	20: // wait reading PAI info completed
		fbCoeReadPAIInfo.bExecute := FALSE;
		IF NOT fbCoeReadPAIInfo.bBusy THEN
			M_UpdateError(fbCoeReadPAIInfo.bError, fbCoeReadPAIInfo.nErrId);
			nStepGetPAIInfo := 0;
		END_IF
END_CASE

fbCoeReadPAIInfo(
	sNetId:= F_CreateAmsNetId(stAdsAddr.netId), 
	nSlaveAddr:= nSlaveAddress, 
	nSubIndex:= 1, 
	nIndex:= nIdxPAIInfo, 
	pDstBuf:= ADR(stPAIInfoData), 
	cbBufLen:= SIZEOF(stPAIInfoData),
	bCompleteAccess:= TRUE);
END_METHOD

METHOD PRIVATE M_WfGetSlaveState : BOOL
// workflow read slave state
CASE nStepGetState OF
	0: // idle
	
	10: // start reading actual slave state
		fbGetSlaveState.bExecute := TRUE;
		nStepGetState := 20;
		
	20: // wait reading actual slave state completed
		fbGetSlaveState.bExecute := FALSE;
		IF NOT fbGetSlaveState.bBusy THEN
			M_UpdateError(fbGetSlaveState.bError, fbGetSlaveState.nErrId);
			IF NOT fbGetSlaveState.bError THEN
				stSlaveState := F_ConvSlaveStateToBitsEx(fbGetSlaveState.state);
			END_IF			
			nStepGetState := 0;				
		END_IF
END_CASE

fbGetSlaveState(
	sNetId := F_CreateAmsNetId(stAdsAddr.netId), 
	nSlaveAddr := nSlaveAddress);
END_METHOD

END_FUNCTION_BLOCK

// ---- POUs/System/Utilities/Convert/F_EcDeviceTimeStampToTime.TcPOU
FUNCTION F_EcDeviceTimeStampToTime : TIME
VAR_INPUT
	nDeviceTimeStamp : ULINT;
END_VAR
VAR
	fDevieTimeStamp : LREAL;
END_VAR

fDevieTimeStamp := ULINT_TO_LREAL(nDeviceTimeStamp) / 1E6; 		// ns to ms
F_EcDeviceTimeStampToTime := LREAL_TO_TIME(fDevieTimeStamp);	// ms to time

END_FUNCTION

// ---- POUs/System/Recipe/FB_RecipeManager.TcPOU
FUNCTION_BLOCK FB_RecipeManager
VAR_IN_OUT	
	/// Recipe	            
	stRecipe	: ST_Settings;
	
	/// Logger
	nLogger		: I_Logger;
	
	/// PlcTag Browser
	fbVar2File	: FB_Var2File;
END_VAR
VAR_INPUT
	/// Directory of recipe files
	sRecipePath					:T_MaxString := '/usr/local/var2file/data/';
	
	/// Allows to load a recipe (Machine is stopped)
	bEnableLoadRecipe			:BOOL;
END_VAR
VAR_OUTPUT
	/// Loading/Saving busy
	bBusy						:BOOL;
	bLoadingBusy				:BOOL;
	stActiveRecipeName			:ST_Text;
	/// Error
	bError						:BOOL;
	stErrorText					:ST_Text;
END_VAR
VAR
	sFileExtension				:STRING := '.csv';
	sObjectNameRecipe			:STRING(255) := 'Services.fbRecipeManager.stRecipeWork';
	
	bInit						:BOOL;
	posSaveCurrent				:R_TRIG;
	posNewRecipe				:R_TRIG;
	posChangeRecipe				:R_TRIG;
	posRefreshRecipeList		:R_TRIG;
	posLoadRecipe				:R_TRIG;
	posDeleteRecipe				:R_TRIG;
	posCopyRecipe				:R_TRIG;

	stRecipeWork				:ST_Settings;
	
	bErrorListRecipes			:BOOL;
	bErrorLoadRecipe			:BOOL;
	bErrorSaveRecipe			:BOOL;
	bErrorCopyRecipe			:BOOL;

	stWorkText					:ST_Text;
	rtrigBusy					:R_TRIG;
END_VAR


// show current recipe data
HMI.stHmi.stOut.stCommon.stRecipe.wsActiveRecipe := stRecipe.stPlant_Settings[E_PlantSettings.ePlantSetting_RecipeName].sValue;
HMI.stHmi.stOut.stCommon.stRecipe.wsActiveRecipeComment := stRecipe.stPlant_Settings[E_PlantSettings.ePlantSetting_RecipeComment].sValue;
HMI.stHmi.stOut.stCommon.stRecipe.wsActiveRecipeProduct := stRecipe.stProduct_Settings[E_ProductSettings.eProductSettings_ProductNumber].sValue;

stActiveRecipeName := F_CreateDynText(stRecipe.stPlant_Settings[E_PlantSettings.ePlantSetting_RecipeName].sValue,0);

// Save current recipe
posSaveCurrent(CLK := stHmi.stIn.stRecipe.bSaveCurrentRecipe);
IF posSaveCurrent.Q AND NOT bBusy THEN
	// copy current
	stRecipeWork := stRecipe;
	M_SaveRecipe(TRUE);
END_IF

// Update current
posChangeRecipe(CLK := stHmi.stIn.stRecipe.bUpdateRecipe );
IF posChangeRecipe.Q THEN
	IF HMI.stHmi.stIn.stRecipe.wsNewEditRecipeName <> "" THEN
		stRecipe.stPlant_Settings[E_PlantSettings.ePlantSetting_RecipeName].sValue := stHmi.stIn.stRecipe.wsNewEditRecipeName;		
	END_IF
	stRecipe.stPlant_Settings[E_PlantSettings.ePlantSetting_RecipeComment].sValue := stHmi.stIn.stRecipe.wsNewEditRecipeComment;		
	stRecipe.stProduct_Settings[E_ProductSettings.eProductSettings_ProductNumber].sValue := stHmi.stIn.stRecipe.wsNewEditRecipeProduct;		
END_IF

// Save as new
posNewRecipe(CLK := stHmi.stIn.stRecipe.bCreateNewRecipe );
IF posNewRecipe.Q AND stHmi.stIn.stRecipe.wsNewEditRecipeName <> "" AND
NOT bBusy THEN
	// copy current
	stRecipeWork := stRecipe;
	// change
	stRecipeWork.stPlant_Settings[E_PlantSettings.ePlantSetting_RecipeName].sValue := stHmi.stIn.stRecipe.wsNewEditRecipeName;		
	stRecipeWork.stPlant_Settings[E_PlantSettings.ePlantSetting_RecipeComment].sValue := stHmi.stIn.stRecipe.wsNewEditRecipeComment;		
	stRecipeWork.stProduct_Settings[E_ProductSettings.eProductSettings_ProductNumber].sValue := stHmi.stIn.stRecipe.wsNewEditRecipeProduct;		
	M_SaveRecipe(TRUE);
END_IF

// refresh list of recipes
posRefreshRecipeList(CLK := stHmi.stIn.stRecipe.bRefreshRecipeList OR NOT bInit);
IF posRefreshRecipeList.Q THEN
	M_ListRecipes(TRUE);
END_IF


// Load
posLoadRecipe(CLK := stHmi.stIn.stRecipe.bLoadSelectedRecipe);
IF posLoadRecipe.Q AND NOT bBusy THEN
	IF stHmi.stIn.stRecipe.nSelectedRecipe >= 0 AND stHmi.stIn.stRecipe.nSelectedRecipe <= CONST.iMaxIdxRecipe AND_THEN 
	HMI.stHmi.stOut.stCommon.stRecipe.aRecipeList[stHmi.stIn.stRecipe.nSelectedRecipe] <> "" THEN
		M_LoadRecipe(TRUE, HMI.stHmi.stOut.stCommon.stRecipe.aRecipeList[stHmi.stIn.stRecipe.nSelectedRecipe]);
	END_IF
END_IF

// delete
posDeleteRecipe(CLK := stHmi.stIn.stRecipe.bDeleteSelectedRecipe);
IF posDeleteRecipe.Q THEN
	IF stHmi.stIn.stRecipe.nSelectedRecipe >= 0 AND stHmi.stIn.stRecipe.nSelectedRecipe <= CONST.iMaxIdxRecipe AND_THEN 
	HMI.stHmi.stOut.stCommon.stRecipe.aRecipeList[stHmi.stIn.stRecipe.nSelectedRecipe] <> "" THEN
		M_DeleteRecipe(TRUE, HMI.stHmi.stOut.stCommon.stRecipe.aRecipeList[stHmi.stIn.stRecipe.nSelectedRecipe]);
	END_IF	
END_IF

// copy
posCopyRecipe(CLK := stHmi.stIn.stRecipe.bCopySelectedRecipe);
IF posCopyRecipe.Q AND NOT bBusy THEN
	IF stHmi.stIn.stRecipe.nSelectedRecipe >= 0 AND stHmi.stIn.stRecipe.nSelectedRecipe <= CONST.iMaxIdxRecipe AND_THEN 
	HMI.stHmi.stOut.stCommon.stRecipe.aRecipeList[stHmi.stIn.stRecipe.nSelectedRecipe] <> "" AND
	stHmi.stIn.stRecipe.wsCopyRecipeNewName <> "" THEN
		M_CopyRecipe(TRUE, 
					HMI.stHmi.stOut.stCommon.stRecipe.aRecipeList[stHmi.stIn.stRecipe.nSelectedRecipe],
					stHmi.stIn.stRecipe.wsCopyRecipeNewName);
	END_IF		
END_IF


// calls
M_SaveRecipe(FALSE);
M_ListRecipes(FALSE);
M_LoadRecipe(FALSE, "");
M_DeleteRecipe(FALSE, "");
M_CopyRecipe(FALSE, "", "");

// Supervision
M_Supervision();

// show HMI Status fields
rtrigBusy(CLK := bBusy);
IF rtrigBusy.Q THEN
	HMI.stHmi.stOut.stCommon.stRecipe.bStatusTextVisible := TRUE; // show immediately
END_IF

IF bError THEN
	HMI.stHmi.stOut.stCommon.stRecipe.stStatusText := stErrorText;
	HMI.stHmi.stOut.stCommon.stRecipe.stStatusColor.color := F_ColorToStringHexColor(STATICS.stColor.Red);
	HMI.stHmi.stOut.stCommon.stRecipe.bStatusTextVisible := TRUE;
	
ELSIF bBusy THEN
	HMI.stHmi.stOut.stCommon.stRecipe.stStatusText := stWorkText;
	HMI.stHmi.stOut.stCommon.stRecipe.stStatusColor.color := F_ColorToStringHexColor(STATICS.stColor.Blue);
	IF Statics.stPulse.bImpulse1000ms THEN
		HMI.stHmi.stOut.stCommon.stRecipe.bStatusTextVisible := NOT HMI.stHmi.stOut.stCommon.stRecipe.bStatusTextVisible;	
	END_IF

ELSE
	HMI.stHmi.stOut.stCommon.stRecipe.bStatusTextVisible := FALSE;
	HMI.stHmi.stOut.stCommon.stRecipe.stStatusText := F_CreateDynText("",0);
	
END_IF


// Enable HMI actions
HMI.stHmi.stOut.stCommon.stRecipe.bEnableSaveCurrentRecipe := NOT bBusy AND HMI.stHmi.stOut.stCommon.stRecipe.wsActiveRecipe <> "";

HMI.stHmi.stOut.stCommon.stRecipe.bEnableCreateNewRecipe := NOT bBusy AND stHmi.stIn.stRecipe.wsNewEditRecipeName <> "";
HMI.stHmi.stOut.stCommon.stRecipe.bEnableUpdateRecipe := NOT bBusy AND stHmi.stIn.stRecipe.wsNewEditRecipeName <> "";

// valid index?
IF stHmi.stIn.stRecipe.nSelectedRecipe >= 0 AND stHmi.stIn.stRecipe.nSelectedRecipe <= CONST.iMaxIdxRecipe THEN
	HMI.stHmi.stOut.stCommon.stRecipe.bEnableLoadRecipe := bEnableLoadRecipe AND
																	NOT bBusy AND 
																	HMI.stHmi.stOut.stCommon.stRecipe.aRecipeList[stHmi.stIn.stRecipe.nSelectedRecipe] <> "";
	HMI.stHmi.stOut.stCommon.stRecipe.bEnableDeleteRecipe := NOT bBusy AND 
																	(HMI.eUserLevel >= E_User_Level.eUser_Level_Maintenance) AND
																	HMI.stHmi.stOut.stCommon.stRecipe.aRecipeList[stHmi.stIn.stRecipe.nSelectedRecipe] <> "" AND
																	HMI.stHmi.stOut.stCommon.stRecipe.aRecipeList[stHmi.stIn.stRecipe.nSelectedRecipe] <> HMI.stHmi.stOut.stCommon.stRecipe.wsActiveRecipe;
	HMI.stHmi.stOut.stCommon.stRecipe.bEnableCopyRecipe := NOT bBusy AND 
																	HMI.stHmi.stOut.stCommon.stRecipe.aRecipeList[stHmi.stIn.stRecipe.nSelectedRecipe] <> "";	
ELSE
	HMI.stHmi.stOut.stCommon.stRecipe.bEnableLoadRecipe := FALSE;
	HMI.stHmi.stOut.stCommon.stRecipe.bEnableDeleteRecipe := FALSE;
	HMI.stHmi.stOut.stCommon.stRecipe.bEnableCopyRecipe := FALSE;	
END_IF



bInit := TRUE;

METHOD PRIVATE M_CopyRecipe : BOOL
VAR_INPUT
	bCopyRecipe				:BOOL;
	wsRecipeName_From		:WSTRING(255);
	wsRecipeName_To			:WSTRING(255);
END_VAR
VAR_INST
	wsRecipeName_FromWork		:WSTRING(255);
	wsRecipeName_ToWork			:WSTRING(255);
	wsRecipeName_ToWork_noExt	:WSTRING(255); //Recipename without FileExtension
	nStep				:INT;
END_VAR

// Reset error
IF HMI.stHmi.stIn.stMain.stButton_Reset.bClick THEN
	bErrorCopyRecipe := FALSE;
END_IF

IF nStep > 0 THEN
	stWorkText := F_CreateDynText("Rezept wird kopiert...",0);
END_IF

CASE nStep OF
	
	0:
		IF bCopyRecipe AND wsRecipeName_From <> "" AND
		wsRecipeName_To <> "" AND NOT fbVar2File.bBusy THEN
			wsRecipeName_FromWork := wsRecipeName_From;
			wsRecipeName_ToWork := wsRecipeName_To;
			wsRecipeName_ToWork_noExt := wsRecipeName_ToWork;
			bErrorCopyRecipe := FALSE;
			bBusy := TRUE;
			nStep := 100;
		END_IF
		
		
		// LOAD

		// load recipe over var2file to stRecipeWork and save it with a new name
		// add sFileExtension ('.csv') to the filename
	100:
		wsRecipeName_FromWork := WCONCAT2x(wsRecipeName_FromWork, TO_WSTRING(sFileExtension));
		wsRecipeName_ToWork := WCONCAT2x(wsRecipeName_ToWork, TO_WSTRING(sFileExtension));
		// copy current for none recipe settings
		stRecipeWork := stRecipe;
		// Load to work
		fbVar2File.M_LoadFromFileRecipe(sRecipePath, TO_STRING(wsRecipeName_FromWork));
		nStep := 110;
		
	110:
		IF fbVar2File.bBusy THEN
			nStep := 120;	
		END_IF
		
	120:
		IF fbVar2File.bError THEN
			bErrorCopyRecipe := TRUE;
			nStep := 200;
			
		ELSIF fbVar2File.bDone THEN
			nStep := 150;
			
		END_IF
		
		
		// SAVE
	150:	
		stRecipeWork.stPlant_Settings[E_PlantSettings.ePlantSetting_RecipeName].sValue := wsRecipeName_ToWork_noExt;
		// Trigger save action
		fbVar2File.M_SaveToFileRecipe(sObjectNameRecipe,
			sRecipePath, TO_STRING(wsRecipeName_ToWork) );
		nStep := 160;
		
	160:
		IF fbVar2File.bBusy THEN
			nStep := 170;	
		END_IF
		
	170:
		IF fbVar2File.bError THEN
			bErrorCopyRecipe := TRUE;
			nStep := 200;
			
		ELSIF fbVar2File.bDone THEN
			nStep := 200;
			
		END_IF
			
	200:
		bBusy := FALSE;
		nStep := 0;
		M_ListRecipes(TRUE);
		
END_CASE
END_METHOD

METHOD PRIVATE M_DeleteRecipe : BOOL
VAR_INPUT
	bDeleteRecipe			:BOOL;
	wsRecipeName			:WSTRING(255);
END_VAR
VAR_INST
	wsRecipeNameWork		:WSTRING(255);
	nStep					:INT;
	fbDeleteFile			:FB_FileDelete;
	
END_VAR

fbDeleteFile.sNetId := '';

IF nStep > 0 THEN
	stWorkText := F_CreateDynText("Rezept wird gelöscht...",0);
END_IF

CASE nStep OF
	
	0:
		IF bDeleteRecipe AND wsRecipeName <> "" THEN
			wsRecipeNameWork := wsRecipeName;
			bBusy := TRUE;
			nStep := 100;
		END_IF
		
		
		// delete recipe
		// add sFileExtension ('.csv') to the filename
	100:
		fbDeleteFile.sPathName := CONCAT4(sRecipePath, sDirSeparator, TO_STRING(wsRecipeNameWork), sFileExtension);
		fbDeleteFile(bExecute := FALSE);
		fbDeleteFile(bExecute := TRUE);
		IF fbDeleteFile.bBusy THEN
			nStep := 110;
		END_IF
		
	110:
		fbDeleteFile(bExecute := FALSE);
		IF NOT fbDeleteFile.bBusy THEN
			nStep := 200;		
		END_IF
		
		// finish
	200:
		bBusy := FALSE;
		nStep := 0;
		M_ListRecipes(TRUE);

END_CASE
END_METHOD

METHOD M_ListRecipes : BOOL
VAR_INPUT
	bRefreshRecipeList			:BOOL;
END_VAR
VAR_INST
	nStepRefreshRecLst			:INT;
	fbListFiles					:FB_EnumFindFileEntry;
	nFileIdx					:INT;
END_VAR

fbListFiles.sNetId := '';
fbListFiles.sPathName := CONCAT4(sRecipePath, sDirSeparator, '*', sFileExtension);

HMI.stHmi.stOut.stCommon.stRecipe.nMaxEntryRecipeList := nFileIdx;

// Reset error
IF HMI.stHmi.stIn.stMain.stButton_Reset.bClick THEN
	bErrorListRecipes := FALSE;
END_IF

CASE nStepRefreshRecLst OF
	
		// wait start
	0:
		fbListFiles( bExecute := FALSE );
		IF bRefreshRecipeList THEN
			FOR nFileIdx := 0 TO CONST.iMaxIdxRecipe DO
				HMI.stHmi.stOut.stCommon.stRecipe.aRecipeList[nFileIdx] := "";
			END_FOR
			nFileIdx := 0;
			bErrorListRecipes := FALSE;
			fbListFiles.eCmd := E_EnumCmdType.eEnumCmd_First;	
			nStepRefreshRecLst := 100;
		END_IF
		
		// Read
	100:
		fbListFiles( bExecute := FALSE );
		fbListFiles( bExecute := TRUE );
		IF fbListFiles.bBusy THEN
			nStepRefreshRecLst := 110;		
		END_IF
		
		// get value
	110:
		fbListFiles( bExecute := FALSE );
		IF NOT fbListFiles.bBusy THEN
			IF NOT fbListFiles.bError THEN
				IF NOT fbListFiles.bEOE AND nFileIdx <= CONST.iMaxIdxRecipe THEN
					// save in array
					HMI.stHmi.stOut.stCommon.stRecipe.aRecipeList[nFileIdx] := TO_WSTRING(F_Replace(fbListFiles.stFindFile.sFileName, sFileExtension, ''));
                    fbListFiles.eCmd := eEnumCmd_Next; (* enum next entry *)
					
					nFileIdx := nFileIdx + 1;
                    nStepRefreshRecLst := 100;
					
				ELSE
					nStepRefreshRecLst := 0; // finish
				END_IF
			
			ELSE
				nStepRefreshRecLst := 0;
				bErrorListRecipes := TRUE;
			END_IF
		END_IF

END_CASE
END_METHOD

METHOD PRIVATE M_LoadRecipe : BOOL
VAR_INPUT
	bLoadRecipe			:BOOL;
	wsRecipeName		:WSTRING(255);
END_VAR
VAR_INST
	wsRecipeNameWork		:WSTRING(255);
	nStep					:INT;
END_VAR

// Reset error
IF HMI.stHmi.stIn.stMain.stButton_Reset.bClick THEN
	bErrorLoadRecipe := FALSE;
END_IF

IF nStep > 0 THEN
	stWorkText := F_CreateDynText("Rezept wird geladen...",0);
END_IF

CASE nStep OF
	
	0:
	
		bLoadingBusy := FALSE;
		IF bLoadRecipe AND wsRecipeName <> "" AND NOT fbVar2File.bBusy THEN
			wsRecipeNameWork := wsRecipeName;
			bBusy := TRUE;
			bLoadingBusy := TRUE;
			bErrorLoadRecipe := FALSE;
			nStep := 100;
		END_IF
		
		
		// load recipe over var2file to stRecipeWork
	100:
		wsRecipeName := WCONCAT2x(wsRecipeNameWork, TO_WSTRING(sFileExtension));
		// copy current for none recipe settings
		stRecipeWork := stRecipe;
		// Trigger load action
		fbVar2File.M_LoadFromFileRecipe(sRecipePath, TO_STRING(wsRecipeName));
		nStep := 110;
		
	110:
		IF fbVar2File.bBusy THEN
			nStep := 120;	
		END_IF
		
	120:
		IF fbVar2File.bError THEN
			bErrorLoadRecipe := TRUE;
			nStep := 200;
			
		ELSIF fbVar2File.bDone THEN
			stRecipe := stRecipeWork; // Takeover recipe data
			nStep := 200;
			
		END_IF
				
	200:
		bBusy := FALSE;
		nStep := 0;

END_CASE
END_METHOD

METHOD M_LoadRecipeStart : BOOL
VAR_INPUT
	wsRecipeName	: WSTRING;
END_VAR
M_LoadRecipe(TRUE, wsRecipeName);
M_LoadRecipeStart := true;
END_METHOD

METHOD PRIVATE M_SaveRecipe : BOOL
VAR_INPUT
	bSaveRecipe			:BOOL;
END_VAR
VAR_INST
	nStep				:INT;
	wsRecipeName		:WSTRING(255);
END_VAR

// Reset error
IF HMI.stHmi.stIn.stMain.stButton_Reset.bClick THEN
	bErrorSaveRecipe := FALSE;
END_IF

IF nStep > 0 THEN
	stWorkText := F_CreateDynText("Rezept wird gespeichert...",0);
END_IF

CASE nStep OF
	
	0:
		wsRecipeName := stRecipeWork.stPlant_Settings[E_PlantSettings.ePlantSetting_RecipeName].sValue;
		IF bSaveRecipe AND wsRecipeName <> "" AND NOT fbVar2File.bBusy THEN
			bBusy := TRUE;
			bErrorSaveRecipe := FALSE;
			nStep := 100;
		END_IF
		
		
		// save recipe over var2file from stRecipeWork
	100:
		wsRecipeName := WCONCAT2x(wsRecipeName, TO_WSTRING(sFileExtension));
		// Trigger save action
		fbVar2File.M_SaveToFileRecipe(sObjectNameRecipe,
			sRecipePath, TO_STRING(wsRecipeName) );
		nStep := 110;
		
	110:
		IF fbVar2File.bBusy THEN
			nStep := 120;	
		END_IF
		
	120:
		IF fbVar2File.bError THEN
			bErrorSaveRecipe := TRUE;
			nStep := 200;
			
		ELSIF fbVar2File.bDone THEN
			nStep := 200;
			
		END_IF
		
	200:
		HMI.stHmi.stOut.stCommon.stRecipe.wsActiveRecipeSavedInfo := TO_WSTRING(Statics.sTimeString);
		bBusy := FALSE;
		nStep := 0;

END_CASE
END_METHOD

METHOD PRIVATE M_Supervision : BOOL
VAR_INPUT
END_VAR
// Error / Status

bError := FALSE;
stErrorText := CONST.stTextListGlobal.stText_notext;

IF bErrorListRecipes THEN
	bError := TRUE;
	stErrorText := CONST.stTextListGlobal.stText_Recipe_ListError;
	
ELSIF bErrorLoadRecipe THEN
	bError := TRUE;
	stErrorText := fbVar2File.stErrorText;
	
ELSIF bErrorSaveRecipe THEN
	bError := TRUE;
	stErrorText := fbVar2File.stErrorText;

ELSIF bErrorCopyRecipe THEN
	bError := TRUE;
	stErrorText := CONST.stTextListGlobal.stText_Recipe_CopyError;
	
END_IF
END_METHOD

END_FUNCTION_BLOCK

// ---- POUs/System/Utilities/Var2File/FB_Var2File.TcPOU
/// Handler for interact with the Var2File tool
FUNCTION_BLOCK FB_Var2File
VAR_INPUT
	stConfig			:ST_Var2File_Config;
END_VAR	
VAR_OUTPUT
	/// Fehlerzustand
	bError				:BOOL;
	/// Fehlertext
	stErrorText			:ST_Text;
	/// Fehlertext Zusatz
	stErrorText_Add		:ST_Text;
	/// Warnung
	bWarning			:BOOL;
	/// Warnungstext
	stWarnText			:ST_Text;

	bBusy		: BOOL;
	bDone		: BOOL;
	nProgress	: UDINT;
END_VAR
VAR
	// object vars
	// start load / save
	fbStart_Exe					: NT_StartProcess;
	// find file
	fbFindFile					: FB_EnumFindFileEntry;
	
	nProcessStep				: INT;

	// Com struct for application
	stAppCom					: ST_Var2File_Com;
	
	// Save to file start flag
	bStartSave2File				: BOOL;
	// load from file flag
	bStartLoadFromFile			: BOOL;
	
	nUseFiltersetId				: INT;
	sUserDynFilterString		: STRING(255);
	sUseFileFolder				: STRING(255);
	sUseFileName				: STRING(255);
	bRecipeMode					: BOOL;
	
	// path to var2file exe
	sPathString					: STRING(100);
	sWriteToPlc					: STRING(5) := 'false';
	sCommand					: T_MAXSTRING;
	
	rtrig_Error					: R_TRIG;
	
	// check communication with var2file tool
	tonCheckCom					: TON;
END_VAR

(*
Parameter:
	-	Mode:			GUI-Mode oder Background-Mode
	-	WriteToPlc:		Funktionsmodus	
		o	wenn TRUE dann werden Variablen in SPS geschrieben
		o	wenn FALSE werden variablen von der SPS in die Datei geschrieben	
	-	AMS-NetID:		Ziel NetId aus der die Variablen gelesen/geschrieben werden sollen
	-	AMS-Port:		Ziel Portnummer
	-	Filter-Set-ID:		ID (Nummer) des Filtersets das angewendet werden soll
	-	Dyn.FilterString:	Statt Filter-Set-ID kann ein Filterstring direkt übergeben werden
	-	FileFolder:		Zielordner für Export-Import Datei
	-	FileName:		Dateiname

Beispiele:
	xxxx.exe -Mode Background -amsnetid “192.168.1.1.1.1” -port 851 -filterset 3
	xxxx.exe -Mode Background -amsnetid “192.168.1.1.1.1” -port 851 -filterstring “GVL_TEST”

	Plausibilität-checks
*)

// now in TC/BSD mode!

tonCheckCom(PT := T#1M);
tonCheckCom.IN := FALSE;

CASE nProcessStep OF
	0:
		// reset data
		IF bStartSave2File OR bStartLoadFromFile THEN
			// reset communication structure
			MEMSET(ADR(stAppCom), 0, SIZEOF(stAppCom));
			
			M_Reset();
			fbStart_Exe.START := FALSE;
			fbFindFile.bExecute := FALSE;
			
			M_CheckPlausibility();
			
			// build path string to exe
			sPathString := CONCAT( stConfig.sAppExeFilePath, stConfig.sAppExeFileName);
		END_IF
		
		// start sequence
		IF bStartSave2File THEN
			sWriteToPlc := 'false';
			bStartSave2File := FALSE;
			nProcessStep := 10; // save data
		ELSIF bStartLoadFromFile THEN
			sWriteToPlc := 'true';
			bStartLoadFromFile := FALSE;
			nProcessStep := 50; // load data
		END_IF
		
// save data
	10: 
		// build command string
		IF stConfig.sAmsNetId = '' THEN
			sCommand := CONCAT4(sPathString, 
						' -mode background ',
						'',
						' -port 851 ');						
		ELSE
			sCommand := CONCAT4(sPathString, 
						' -mode background -amsNetId "',
						stConfig.sAmsNetId,
						'" -port 851 ');			
		END_IF

		// add filter
		IF nUseFiltersetId <> 0 THEN
			sCommand := CONCAT3(sCommand, 
						' -filterSet ',
						INT_TO_STRING(nUseFiltersetId));
		ELSE
			sCommand := CONCAT4(sCommand, 
						' -filterstring "',
						sUserDynFilterString,
						'"');
		END_IF
		
		// recipe mode
		IF bRecipeMode THEN
			sCommand := CONCAT3(sCommand, 
						' -recipe true ',
						'');			
		END_IF
				
		// add file destination
		sCommand := CONCAT5(sCommand, 
					' -filePath "',
					sUseFileFolder,
					'" -fileName ',
					sUseFileName);
	
		nProcessStep := 100;
		
// load data
	50: // enum first entry
		fbFindFile.eCmd := eEnumCmd_First;
		nProcessStep := 60;
		
	60: // start search file
		fbFindFile(bExecute := FALSE);
		fbFindFile(bExecute := TRUE);
		nProcessStep := 70;
		
	70: // wait search is done
		fbFindFile.bExecute := FALSE;
		IF NOT fbFindFile.bBusy THEN
			IF NOT fbFindFile.bError THEN
				// File found
				IF fbFindFile.stFindFile.sFileName = sUseFileName THEN
					nProcessStep := 80;
					
				// End of file reached -> file not found
				ELSIF fbFindFile.bEOE THEN
					bError := TRUE;
					stErrorText := F_CreateDynText(TO_WSTRING(CONCAT(sUseFileName, ' - file not found!')), 0);
				
					bBusy := FALSE;
					nProcessStep := 0;
					
				// search next file
				ELSE
					fbFindFile.eCmd := eEnumCmd_Next; // enum next entry 
					nProcessStep := 60;
				END_IF
				
			// log error
			ELSE
				bError := TRUE;
				stErrorText := F_CreateDynText(TO_WSTRING(CONCAT(sUseFileName, ' - file or directory not found!')), 0);
							
				bBusy := FALSE;
				nProcessStep := 0;
			END_IF
		END_IF

	80: 
		// build command string
		IF stConfig.sAmsNetId = '' THEN
			sCommand := CONCAT4(sPathString, 
						' -mode background -writeToPlc true ',
						'',
						' -port 851 ');		
		ELSE
			sCommand := CONCAT4(sPathString, 
						' -mode background -writeToPlc true -amsNetId "',
						stConfig.sAmsNetId,
						'" -port 851 ');			
		END_IF
		
		// recipe mode
		IF bRecipeMode THEN
			sCommand := CONCAT3(sCommand, 
						' -recipe true ',
						'');			
		END_IF
			
		// add file destination
		sCommand := CONCAT6(sCommand, 
					' -filePath "',
					sUseFileFolder,
					'" -fileName "',
					sUseFileName,
					'"');
					
		nProcessStep := 100;

// start application and check communication with tool

	100: // execute app
		fbStart_Exe.START := TRUE;
		// wait busy
		IF fbStart_Exe.BUSY THEN
			fbStart_Exe.START := FALSE;
			nProcessStep := 110;
		END_IF
		
	110: // wait not busy
		IF NOT fbStart_Exe.BUSY THEN
			IF fbStart_Exe.ERR THEN
				bBusy := FALSE;
				nProcessStep := 0;
			ELSE
				nProcessStep := 120;
			END_IF
		END_IF
	
	120: // check communication with tool
		// tool is done
		IF stAppCom.bAppJobFinished OR stAppCom.nAppProgress = 100 THEN
			M_ErrorCode(stAppCom.nAppErrorCode);
			bBusy := FALSE;
			nProcessStep := 0;
			bRecipeMode := FALSE;
		ELSE
			tonCheckCom.IN := stAppCom.nAppProgress = 0;
		END_IF
		
		// error -> no communication
		IF tonCheckCom.Q OR stAppCom.nAppErrorCode > 0 THEN
			// create alarm
			bError := TRUE;
			stErrorText := F_CreateDynText(WCONCAT2x("Error Var2File tool. Error: ", M_ErrorCode(stAppCom.nAppErrorCode)), 0);
			bBusy := FALSE;
			nProcessStep := 0;
			bRecipeMode := FALSE;
		END_IF
		
END_CASE

// call FB's
IF nProcessStep > 0 THEN
	fbStart_Exe(
			NETID	:= '', // local
			PATHSTR	:= '/bin/sh', // now in TC/BSD mode!, sPathString,
			DIRNAME	:= '/usr/local/var2file', // stConfig.sAppExeFilePath,
			COMNDLINE := CONCAT4('ExecuteVar2File.sh ', sWriteToPlc, ' ', sUseFileName), //sCommand,
			TMOUT	:= T#5S,
			BUSY	=> , 
			ERR		=> , 
			ERRID	=> );
			
	fbFindFile(
			sNetID := '', 
			sPathName := CONCAT3(sUseFileFolder, sDirSeparator, '*.*'),
			tTimeout := T#5S);
END_IF	
						
// set alarm
rtrig_Error( CLK := fbStart_Exe.ERR);
IF rtrig_Error.Q THEN
	bError := TRUE;
	stErrorText := F_CreateDynText(WCONCAT2x("Var2File NT_Process ErrorID: ", TO_WSTRING(fbStart_Exe.ERRID)), 0);
END_IF

bDone := stAppCom.bAppJobFinished AND NOT bBusy;
nProgress := stAppCom.nAppProgress;

			
(*// call FB's (nur Backup hier)
fbStart_Var2File(
			NETID	:= '', 
			PATHSTR	:= 'C:\Rmth\Software\var2file\var2file.exe',//'C:\Tools\var2file_Rmth\PlcTag.WinForms.App.exe', //sPathString, 
			DIRNAME	:= 'C:\Rmth\Software\var2file',//'C:\Tools\var2file_Rmth', //WSTRING_TO_STRING(wsUseFileFolder), 
			COMNDLINE := 'C:\Rmth\Software\var2file\var2file.exe -mode background -amsNetId "192.168.163.1.1.1" -port 851 -filterSet 1 -filePath "C:\Temp" -fileName PlcData.json', 
			TMOUT	:= T#5S,
			BUSY	=> , 
			ERR		=> , 
			ERRID	=> );*)

METHOD PROTECTED M_CheckPlausibility : BOOL
VAR_INPUT
END_VAR
VAR
	bPlausible			: BOOL;
	nLastBackslashPos	: INT;
END_VAR
// set marker bit
bPlausible := FALSE;

// plausibility check
IF stConfig.sAppExeFilePath = '' THEN
	bError := TRUE;
	stErrorText := F_CreateDynText("No Var2File exe path", 0);
	
ELSIF stConfig.sAppExeFileName = '' THEN
	bError := TRUE;
	stErrorText := F_CreateDynText("No Var2File exe name", 0);
	
ELSIF sUseFileFolder = '' THEN
	bError := TRUE;
	stErrorText := F_CreateDynText("No file folder selected (Var2File)", 0);
	
ELSIF sUseFileName = '' THEN
	bError := TRUE;
	stErrorText := F_CreateDynText("No file name selected (Var2File)", 0);
	
ELSE
	bPlausible := TRUE;
	
	// check if there is 'no' backslash at the end of the file directory path
	IF RIGHT(sUseFileFolder, 1) = sDirSeparator THEN
		nLastBackslashPos := LEN(sUseFileFolder);
		sUseFileFolder := DELETE(sUseFileFolder, 1, nLastBackslashPos);
	END_IF
	
	// no point found in the filename (assumption no file extension)
	IF FIND(sUseFileName, '.') = 0 THEN
		// add file extension .json
		sUseFileName := CONCAT(sUseFileName, '.json');
	END_IF
	
	// check if there is a backslash at the end of the exe directory path
	IF RIGHT(stConfig.sAppExeFilePath, 1) <> sDirSeparator THEN
		stConfig.sAppExeFilePath := CONCAT(stConfig.sAppExeFilePath, sDirSeparator);
	END_IF
END_IF

IF NOT bPlausible THEN
	// reset start signals
	bStartSave2File := FALSE;
	bStartLoadFromFile := FALSE;
	bBusy := FALSE;
END_IF

M_CheckPlausibility := TRUE;
END_METHOD

/// convert Var2File error code into an text and send alarm
METHOD PRIVATE M_ErrorCode : WSTRING
VAR_INPUT
	/// Applications error code
	nErrorCode			: UDINT;
END_VAR

CASE nErrorCode OF
	0:	// No error
		RETURN;
		
	100:
		M_ErrorCode := "Job canceled by plc";
		
	101:
		M_ErrorCode := "Job canceled by operator";
		
	1000:
		M_ErrorCode := "Reading plc tags failed";
		
	1001:
		M_ErrorCode := "Reading plc tag values failed";
		
	1002:
		M_ErrorCode := "Reading backup file failed";
		
	1003:
		M_ErrorCode := "Writing backup file failed";
		
	1004:
		M_ErrorCode := "Writing plc tag values failed";
		
	ELSE
		M_ErrorCode := WCONCAT2x("Undefined error code: Error ID = ", TO_WSTRING(nErrorCode));
END_CASE

// create alarm
bError := TRUE;
END_METHOD

/// cancel active job
METHOD M_JobCancel : BOOL
VAR_INPUT
END_VAR

// not allowed if not running
IF nProcessStep <= 0 THEN
	RETURN;
END_IF

stAppCom.bJobCancelRequest := TRUE;
END_METHOD

/// Starts the var2file tool with the given file name
METHOD M_LoadFromFile : BOOL
VAR_INPUT
	sFileName					: STRING(255);	
END_VAR
// not allowed if already running
IF bBusy THEN
	M_LoadFromFile := FALSE;
	RETURN;
END_IF

M_LoadFromFile := M_LoadFromFileEx(stConfig.sDefaultFileFolderPath, sFileName);
END_METHOD

/// Starts the var2file tool with the given file folder and name
METHOD M_LoadFromFileEx : BOOL
VAR_INPUT
	sFileFolder					: STRING(255);
	sFileName					: STRING(255);	
END_VAR
// not allowed if already running
IF bBusy THEN
	M_LoadFromFileEx := FALSE;
	RETURN;
END_IF

nUseFiltersetId := 0;
sUserDynFilterString := '';

sUseFileFolder	:= sFileFolder;
sUseFileName := sFileName;

bStartLoadFromFile := TRUE;

bBusy := TRUE;

M_LoadFromFileEx := TRUE;
END_METHOD

/// Starts the var2file tool with the given file folder and name
METHOD M_LoadFromFileRecipe : BOOL
VAR_INPUT
	sFileFolder					: STRING(255);
	sFileName					: STRING(255);	
END_VAR
// not allowed if already running
IF bBusy THEN
	M_LoadFromFileRecipe := FALSE;
	RETURN;
END_IF

nUseFiltersetId := 0;
sUserDynFilterString := '';

sUseFileFolder	:= sFileFolder;
sUseFileName := sFileName;
bRecipeMode := TRUE;

bStartLoadFromFile := TRUE;

bBusy := TRUE;

M_LoadFromFileRecipe := TRUE;
END_METHOD

METHOD M_Reset : BOOL
VAR_INPUT
END_VAR
/// Fehlerzustand
bError := FALSE;
/// Fehlertext
stErrorText := CONST.stTextListGlobal.stText_notext;
/// Fehlertext Zusatz
stErrorText_Add	:= CONST.stTextListGlobal.stText_notext;
/// Warnung
bWarning := FALSE;
/// Warnungstext
stWarnText := CONST.stTextListGlobal.stText_notext;
END_METHOD

/// Starts the var2file tool for all user variables
METHOD M_SaveToFileAll : BOOL
VAR_INPUT
	sFileName					: STRING(255);	
END_VAR
// not allowed if already running
IF bBusy THEN
	M_SaveToFileAll := FALSE;
	RETURN;
END_IF

M_SaveToFileAll := M_SaveToFileFilterSetEx(stConfig.nFilterSetIDAllVars, stConfig.sDefaultFileFolderPath, sFileName);
END_METHOD

/// Starts the var2file tool with the given filterset
METHOD M_SaveToFileFilterSet : BOOL
VAR_INPUT
	nFiltersetId				: INT;
	sFileName					: STRING(255);	
END_VAR
// not allowed if already running
IF bBusy THEN
	M_SaveToFileFilterSet := FALSE;
	RETURN;
END_IF

M_SaveToFileFilterSet := M_SaveToFileFilterSetEx(nFiltersetId, stConfig.sDefaultFileFolderPath, sFileName);
END_METHOD

/// Starts the var2file tool with the given filterset
METHOD M_SaveToFileFilterSetEx : BOOL
VAR_INPUT
	nFiltersetId				: INT;
	sFileFolder					: STRING(255);
	SFileName					: STRING(255);	
END_VAR
// not allowed if already running
IF bBusy OR nFiltersetId = 0 THEN
	M_SaveToFileFilterSetEx := FALSE;
	RETURN;
END_IF

nUseFiltersetId := nFiltersetId;
sUserDynFilterString := '';
bRecipeMode := FALSE;

sUseFileFolder	:= sFileFolder;
sUseFileName := sFileName;

bStartSave2File := TRUE;

bBusy := TRUE;

M_SaveToFileFilterSetEx := TRUE;
END_METHOD

/// Starts the var2file tool with the given filterstring
METHOD M_SaveToFileFilterString : BOOL
VAR_INPUT
	sDynFilterString			: STRING(255);
	sFileName					: STRING(255);	
END_VAR
// not allowed if already running
IF bBusy THEN
	M_SaveToFileFilterString := FALSE;
	RETURN;
END_IF

M_SaveToFileFilterString := M_SaveToFileFilterStringEx(sDynFilterString, stConfig.sDefaultFileFolderPath, sFileName);
END_METHOD

/// Starts the var2file tool with the given filterstring
METHOD M_SaveToFileFilterStringEx : BOOL
VAR_INPUT
	sDynFilterString			: STRING(255);
	sFileFolder					: STRING(255);
	sFileName					: STRING(255);	
END_VAR
// not allowed if already running
IF bBusy OR sDynFilterString = '' THEN
	M_SaveToFileFilterStringEx := FALSE;
	RETURN;
END_IF

nUseFiltersetId := 0;
sUserDynFilterString := sDynFilterString;
bRecipeMode := FALSE;

sUseFileFolder	:= sFileFolder;
sUseFileName := sFileName;

bStartSave2File := TRUE;

bBusy := TRUE;

M_SaveToFileFilterStringEx := TRUE;
END_METHOD

METHOD M_SaveToFileRecipe : BOOL
VAR_INPUT
	sDynFilterString			: STRING(255) := 'Objects.fbRecipeManager.stRecipe.stRecipeWork';
	sFileFolder					: STRING(255);
	sFileName					: STRING(255);	
END_VAR
// not allowed if already running
IF bBusy OR sDynFilterString = '' THEN
	M_SaveToFileRecipe := FALSE;
	RETURN;
END_IF

nUseFiltersetId := 0;
sUserDynFilterString := sDynFilterString;
bRecipeMode := TRUE;

sUseFileFolder	:= sFileFolder;
sUseFileName := sFileName;

bStartSave2File := TRUE;

bBusy := TRUE;

M_SaveToFileRecipe := TRUE;
END_METHOD

END_FUNCTION_BLOCK

// ---- POUs/System/Utilities/String/WConcat2x.TcPOU
FUNCTION WConcat2x : WSTRING(255)
VAR_INPUT
	wsExpression1: WSTRING(255);
	wsExpression2: WSTRING(255);
END_VAR

WConcat2x := WCONCAT(wsExpression1, wsExpression2);

END_FUNCTION

// ---- POUs/System/Utilities/String/F_Replace.TcPOU
FUNCTION F_Replace : STRING(255)
VAR_INPUT
	sInputText		:STRING(255);
	sSearchText		:STRING(255);
	sReplaceText	:STRING(255);
END_VAR
VAR
	idxFnd			:INT;
	iLength			:INT;
END_VAR

idxFnd := FIND(sInputText, sSearchText);
iLength := LEN(sSearchText);

IF idxFnd > 0 THEN
	F_Replace := REPLACE(sInputText, sReplaceText, iLength, idxFnd);
ELSE
	F_Replace := sInputText;
END_IF

END_FUNCTION

// ---- POUs/Plant/M001_Module/FB_M001_Module.TcPOU
FUNCTION_BLOCK FB_M001_Module EXTENDS FB_ModuleBase
VAR
	// module components

	
	// actor UIs, access to: iStatus, fPosition, iVisibleState, ..
	
	// IO ref
	stIO			: REFERENCE TO ST_M001_IO;
	
	// instannce var's
	
	

END_VAR

/// 
/// Module 001 function block 
///

METHOD PRIVATE GetHgCmd_Default : ST_St030_Command
VAR
	result : ST_St030_Command;
END_VAR
// get next job for handling
// 1. drop existing HG pallet
// 2/3. put empty pallet to storage 1/2
// 4/5. put unfinished pallet to storage 1/2

// chk HG has active command
IF Plant.stSt030IHandling.ActiveCommand.Command <> E_St030_Command.eSt030_Command_none THEN
	// sb.Set('wait for active HG command done. Active cmd: ')
		//	 .Append(TO_String(Plant.stSt030IHandling.ActiveCommand.Command));
	RETURN;
END_IF
	
// prio 1: put handling command (e.g. drop existing pallet)
result := GetHgCmd_Default_Put();
IF result.Command <> E_St030_Command.eSt030_Command_none THEN
	// sb.Set('wait for requested HG command is active, cmd: ')
		//	 .Append(TO_String(Plant.stSt030IHandling.CommandRequest.Command));
	GetHgCmd_Default := result;
	RETURN;
END_IF

// prio 2-6: get handling command (e.g. get unfinished pallet)
result := GetHgCmd_Default_Get();
GetHgCmd_Default := result;
END_METHOD

METHOD PRIVATE GetHgCmd_Default_Get : ST_St030_Command
VAR
	none	: ST_St030_Command;
END_VAR
// default logic
GetHgCmd_Default_Get := none;

// chk pallet already on handling
IF Plant.stSt030IHandling.Pallet.CarrierPresent THEN
	RETURN;
END_IF

// prio 2: req empty carrier @ storage #1
IF Plant.stSt050IMould.bReqS1Empty AND 
NOT Plant.stSt040IStorage.Pallet1.HasEmptyWorkpieceplaces THEN
	IF Plant.stSt040IStorage.Pallet1.CarrierPresent THEN
		GetHgCmd_Default_Get := GetHgCmd_StorageGet(1); // 1st, get pallet from storage 1
	ELSE
		// sb.Set('wait for oven 1/2 has empty pallet)
		GetHgCmd_Default_Get := GetHgCmd_OvenGetEmptyPallet(); // get empty pallet from oven A/B
	END_IF
	RETURN;
END_IF

// prio 3: req empty carrier @ storage #2
IF Plant.stSt050IMould.bReqS2Empty AND 
NOT Plant.stSt040IStorage.Pallet2.HasEmptyWorkpieceplaces THEN
	IF Plant.stSt040IStorage.Pallet2.CarrierPresent THEN
		GetHgCmd_Default_Get := GetHgCmd_StorageGet(2); // 1st, get pallet from storage 2
	ELSE
		// sb.Set('wait for oven 1/2 has empty pallet)
		GetHgCmd_Default_Get := GetHgCmd_OvenGetEmptyPallet(); // get empty pallet from oven A/B
	END_IF
	RETURN;
END_IF

// prio 4: req unfinished carrier @ storage #1
IF Plant.stSt050IMould.bReqS1Unfinished AND 
NOT Plant.stSt040IStorage.Pallet1.HasWorkpiecesWithRequestStatus THEN
	IF Plant.stSt040IStorage.Pallet1.CarrierPresent THEN
		GetHgCmd_Default_Get := GetHgCmd_StorageGet(1); // 1st, get pallet from storage 1
	ELSE
		// sb.Set('wait for oven 1/2 has unfinished pallet)
		GetHgCmd_Default_Get := GetHgCmd_OvenGetUnfinishedPallet(); // get unfinished pallet from oven A/B
	END_IF
	RETURN;
END_IF

// prio 5: req unfinished carrier @ storage #2
IF Plant.stSt050IMould.bReqS2Unfinished AND 
NOT Plant.stSt040IStorage.Pallet2.HasWorkpiecesWithRequestStatus THEN
	IF Plant.stSt040IStorage.Pallet2.CarrierPresent THEN
		GetHgCmd_Default_Get := GetHgCmd_StorageGet(2); // 1st, get pallet from storage 2
	ELSE
		// sb.Set('wait for oven 1/2 has unfinished pallet)
		GetHgCmd_Default_Get := GetHgCmd_OvenGetUnfinishedPallet(); // get unfinished pallet from oven A/B
	END_IF
	RETURN;
END_IF

// prio 6: req no carrier @ storage #1/2
IF (Plant.stSt050IMould.bReqS1NoCarrier OR Plant.stM001IModule.bEmptyPlant) AND Plant.stSt040IStorage.Pallet1.CarrierPresent THEN
	GetHgCmd_Default_Get := GetHgCmd_StorageGet(1); // empty plant, get pallet from storage 1
ELSIF (Plant.stSt050IMould.bReqS2NoCarrier OR Plant.stM001IModule.bEmptyPlant) AND Plant.stSt040IStorage.Pallet2.CarrierPresent THEN
	GetHgCmd_Default_Get := GetHgCmd_StorageGet(2); // empty plant, get pallet from storage 2
END_IF
END_METHOD

METHOD PRIVATE GetHgCmd_Default_Put : ST_St030_Command
VAR
	none,
	result	: ST_St030_Command;
END_VAR
// default logic
GetHgCmd_Default_Put := none;

// chk pallet on handling
IF NOT Plant.stSt030IHandling.Pallet.CarrierPresent THEN
	RETURN;
END_IF

// unfinished @ hg --> to storage 1/2
IF Plant.stSt030IHandling.Pallet.HasUnfinishedWorkpieces THEN
	// sb.Set('wait for storage request unfinished')
	IF Plant.stSt050IMould.bReqS1Unfinished AND
	   NOT Plant.stSt040IStorage.Pallet1.CarrierPresent THEN
		GetHgCmd_Default_Put := GetHgCmd_StationPut(E_Station.eStation_ST040_Storage, 1);
	ELSIF Plant.stSt050IMould.bReqS2Unfinished AND
	   NOT Plant.stSt040IStorage.Pallet2.CarrierPresent THEN
		GetHgCmd_Default_Put := GetHgCmd_StationPut(E_Station.eStation_ST040_Storage, 2);
	ELSE
		// unfinished back to oven 1/2
		GetHgCmd_Default_Put := GetHgCmd_StationPut(Plant.stSt030IHandling.Source);
	END_IF
	RETURN;
END_IF

// empty @ hg --> to storage 1/2
IF Plant.stSt030IHandling.Pallet.HasEmptyWorkpieceplaces THEN
	// sb.Set('wait for storage request empty')
	IF Plant.stSt050IMould.bReqS1Empty AND
	   NOT Plant.stSt040IStorage.Pallet1.CarrierPresent THEN
		GetHgCmd_Default_Put := GetHgCmd_StationPut(E_Station.eStation_ST040_Storage, 1);
	ELSIF Plant.stSt050IMould.bReqS2Empty AND
	   NOT Plant.stSt040IStorage.Pallet2.CarrierPresent THEN
		GetHgCmd_Default_Put := GetHgCmd_StationPut(E_Station.eStation_ST040_Storage, 2);
	ELSE
		// empty back to oven 1/2
		GetHgCmd_Default_Put := GetHgCmd_StationPut(Plant.stSt030IHandling.Source);
	END_IF
	RETURN;
END_IF 

// finished & pallet full @ hg --> to oven 2
IF Plant.stSt030IHandling.Pallet.HasAllWorkpiecesFinished THEN
	// sb.Set('wait for oven 2 rdy for finished pallet)
	// full back to oven 1/2
	GetHgCmd_Default_Put := GetHgCmd_StationPut(Plant.stSt030IHandling.Source);
END_IF

//sb.Set('state not implemented: no empty/finished or unfinished');
END_METHOD

METHOD PRIVATE GetHgCmd_OvenGetEmptyPallet : ST_St030_Command
VAR
	result : ST_St030_Command;
END_VAR
result.Command := E_St030_Command.eSt030_Command_none;
IF Plant.stSt010IOvenA.Trolley.HasCarrierWithEmptyWorkpieceplace THEN
	result.Command := E_St030_Command.eSt030_Command_OvenA_Get; // get empty pallet from oven A
	result.Position := Plant.stSt010IOvenA.Trolley.SlotOfCarrierWithEmptyWorkpieceplace; 
ELSIF Plant.stSt020IOvenB.Trolley.HasCarrierWithEmptyWorkpieceplace THEN
	result.Command := E_St030_Command.eSt030_Command_OvenB_Get; // get empty pallet from oven B
	result.Position := Plant.stSt020IOvenB.Trolley.SlotOfCarrierWithEmptyWorkpieceplace;
END_IF

GetHgCmd_OvenGetEmptyPallet := result;
END_METHOD

METHOD PRIVATE GetHgCmd_OvenGetUnfinishedPallet : ST_St030_Command
VAR
	result : ST_St030_Command;
END_VAR
result.Command := E_St030_Command.eSt030_Command_none;
IF Plant.stSt010IOvenA.Trolley.HasCarrierWithUnfinishedWorkpiece THEN
	result.Command := E_St030_Command.eSt030_Command_OvenA_Get; // get unfinished pallet from oven A
	result.Position := Plant.stSt010IOvenA.Trolley.SlotOfCarrierWithUnfinishedWorkpiece;	
ELSIF Plant.stSt020IOvenB.Trolley.HasCarrierWithUnfinishedWorkpiece THEN
	result.Command := E_St030_Command.eSt030_Command_OvenB_Get; // get unfinished pallet from oven B
	result.Position := Plant.stSt020IOvenB.Trolley.SlotOfCarrierWithUnfinishedWorkpiece;
END_IF

GetHgCmd_OvenGetUnfinishedPallet := result;
END_METHOD

METHOD PRIVATE GetHgCmd_StationPut : ST_St030_Command
VAR_INPUT
	eStation 	: E_Station;
	iIxd 		: INT := 0;
END_VAR
VAR
	result 		: ST_St030_Command;
END_VAR
CASE eStation OF
	E_Station.eStation_ST010_OvenA:
		IF Plant.stSt010IOvenA.Trolley.HasEmptySlot THEN
			result.Command := E_St030_Command.eSt030_Command_OvenA_Put;
			result.Position := Plant.stSt010IOvenA.Trolley.EmptySlot;
		ELSE
			ModuleWarning.ArgSbAppend('Station has no empty slot')
				 .ArgSbAppendS(TO_STRING(eStation))
				 .ArgSetSbRaise();		
		END_IF
		
	E_Station.eStation_ST020_OvenB:
		IF Plant.stSt020IOvenB.Trolley.HasEmptySlot THEN
			result.Command := E_St030_Command.eSt030_Command_OvenB_Put;
			result.Position := Plant.stSt020IOvenB.Trolley.EmptySlot;
		ELSE
			ModuleWarning.ArgSbAppend('Station has no empty slot')
				 .ArgSbAppendS(TO_STRING(eStation))
				 .ArgSetSbRaise();	
		END_IF
		
	E_Station.eStation_ST040_Storage:
		result.Command := E_St030_Command.eSt030_Command_Storage_Put;
		result.Position := iIxd;
		
ELSE
	ModuleWarning.ArgSbAppend('Put to station not implemented! Station: ')
				 .ArgSbAppendS(TO_STRING(eStation))
				 .ArgSetSbRaise();
END_CASE

GetHgCmd_StationPut := result;
END_METHOD

METHOD PRIVATE GetHgCmd_StorageGet : ST_St030_Command
VAR_INPUT
	iIxd : INT;
END_VAR
VAR
	result : ST_St030_Command;
END_VAR
result.Command := E_St030_Command.eSt030_Command_Storage_Get;
result.Position := iIxd;

GetHgCmd_StorageGet := result;
END_METHOD

METHOD PRIVATE GetHgCmd_Type3 : ST_St030_Command
VAR
	none : ST_St030_Command;
END_VAR

// hg logic 3

GetHgCmd_Type3 := none;


// e.g.: impelemt custom handling command for type 3...
END_METHOD

METHOD PRIVATE GetHgCmd_Type5 : ST_St030_Command
VAR
	none : ST_St030_Command;
END_VAR

// hg logic 5

GetHgCmd_Type5 := none;


// e.g.: impelemt custom handling command for type 5...
END_METHOD

METHOD PRIVATE GetHgCmd_Type6 : ST_St030_Command
VAR
	none : ST_St030_Command;
END_VAR

// hg logic 6

GetHgCmd_Type6 := none;


// e.g.: impelemt custom handling command for type 6...
END_METHOD

METHOD PROTECTED M_CallObjects : BOOL
VAR
END_VAR

CALL_BVS();

// call..
END_METHOD

METHOD INTERNAL M_DynManual : BOOL
VAR_INPUT
END_VAR
IF NOT bInitManual THEN
	bInitManual := TRUE;
	MEMSET(ADR(stHmiManualOut.stObjects), 0, SIZEOF(stHmiManualOut.stObjects)); // reset
	
	//M_InitDynManualUi(fbAxisVmUi);
	
	//fbAxisVmUi.M_TargetListClear();
	//fbAxisVmUi.M_TargetListAddItem(F_CreateDynText("Home pos", 0), 15);
	//fbAxisVmUi.M_TargetListAddItem(F_CreateDynText("Pos Service", 0), 100);
END_IF
END_METHOD

METHOD PROTECTED M_DynMonitoring : BOOL
VAR_INPUT
END_VAR
M_DynMonitoring := SUPER^.M_DynMonitoring();

// init
IF NOT bInitMonitoring THEN
	bInitMonitoring := TRUE;
	MEMSET(ADR(stLocalMonitoring), 0, SIZEOF(stLocalMonitoring)); // reset
	
	M_InitDynMonitoringItem(0, 								// monitoring index 
							"VM Position", 					// name
							Name, 							// group (station name)
							E_DataType.eDataType_lreal, 	// data type							
							stTextListGlobal.stText_m);		// unit	

	M_InitDynMonitoringItem(1, "VM Geschwindigkeit", Name, E_DataType.eDataType_lreal, stTextListGlobal.stText_mmin);
END_IF

//stLocalMonitoring.astMonitoring[0].fValue := stM001IModule.fVmPos;
//stLocalMonitoring.astMonitoring[1].fValue := stM001IModule.fVmSpeed;
END_METHOD

METHOD INTERNAL M_DynSettings : BOOL
VAR_INST
	fSpeedMir : LREAL;
END_VAR
// init station settings
IF NOT bInitSettings THEN
	bInitSettings := TRUE;
	stLocalSettingsBackup := stLocalSettings; // backup
	MEMSET(ADR(stLocalSettings), 0, SIZEOF(stLocalSettings)); // reset
	
	M_InitDynSettingsItem(E_M001_Settings.eM001_Settings_Deaktiv,		// settings index
		TO_WSTRING(E_M001_Settings.eM001_Settings_Deaktiv),				// settings wsIndex
		Name,															// group
		stTextListGlobal.stText_DeactivateModule,						// name
		stTextListGlobal.stText_bool, E_DataType.eDataType_bool,		// unit & data type
		0, 1, 6);														// min, max & user level

	M_InitDynSettingsItem(E_M001_Settings.eM001_Settings_Autohome,
		TO_WSTRING(E_M001_Settings.eM001_Settings_Autohome),
		Name,
		stTextListGlobal.stText_AutoHome,
		stTextListGlobal.stText_bool, E_DataType.eDataType_bool,
		0, 1, 3);
		
//	M_InitDynSettingsItem(E_M001_Settings.eM001_Settings_PalletLayout,
//		TO_WSTRING(E_M001_Settings.eM001_Settings_PalletLayout),
//		Name,
//		F_CreateDynTextDefault("Palettenlayout (1-4)"),
//		stTextListGlobal.stText_notext, E_DataType.eDataType_int,
//		1, 4, 3);
		
	// restore values
	F_RestoreSettingValues(stLocalSettings.stDynStationSettings, stLocalSettingsBackup.stDynStationSettings);
END_IF

// run settings mgmt
//F_Settings_Management(stLocalSettings.stDynStationSettings);

// map current settings values
bAutoHome := stLocalSettings.stDynStationSettings[E_M001_Settings.eM001_Settings_Autohome].bValue;
END_METHOD

METHOD INTERNAL M_Fast : BOOL
VAR_INPUT
END_VAR
// fast task

Plant.fbSt030Handling.M_SequenceSearch();
//Plant.fbSt050Mould.M_Run();
END_METHOD

METHOD PROTECTED M_Homing
VAR
	bTmp : BOOL;
	stTmpTxt : ST_Text;
END_VAR
// Homing sequence
CASE sqHome.Step OF
	
	0:	
		sqHome.Info.Set("Warte auf GRST Start");
		IF RunStep AND NOT sqHome.InHome AND bRunHoming THEN
			bBusy := TRUE;
			sqAuto.Step := 0;
			sqHome.StartSequence()
				  .Step := 10;
		END_IF

	10:
		sqHome.Info.Set("Grundstellungsfahrt aktiv");
		IF P_Safety.bMachineRequestStop THEN
			sqHome.Info.Set("Anforderung Stop aktiv");
		ELSIF NOT P_Safety.SafetyOk THEN
			sqHome.Info.Set("Sicherheit nicht ok");
		ELSIF bRunHoming THEN
			sqHome.Step := 20;
		END_IF	
	
	20:
		sqHome.Info.Set("Warte auf Stationen in GRST");
		bTmp := TRUE;
		//FOR ii := 0 TO E_Station.eStation_nMaxIdx DO
		//	IF aIStaton[ii] = 0 THEN
		//		CONTINUE;
		//	END_IF
		//	IF NOT aIStaton[ii].InHome THEN
		//		stTmpTxt := aIStaton[ii].Name;
		//		sqHome.Info.Set("Warte auf Station in GRST: ")
		//				   .Append(stTmpTxt.wsName);
		//		bTmp := FALSE;
		//		EXIT;
		//	END_IF
		//END_FOR
		IF bTmp THEN			
			sqHome.Step := 100;
		END_IF
		
	100:
		sqHome.Info.Set("Grundstellungsfahrt aktiv");
		sqHome.Step := 1000;

	//	homing done			
	1000:
		sqHome.Info.Set("Grundstellung erreicht");
		IF sqHome.StepTime > T#1S THEN			
			bBusy := FALSE;
			sqHome.InHome := TRUE;
			bStopped := TRUE;
			bRunHoming := FALSE;
			sqAuto.Step := 0;
			sqHome.StopSequence()
				  .Step := 0;
		END_IF
END_CASE
END_METHOD

METHOD PUBLIC M_Init : IModule
VAR_INPUT
END_VAR
VAR
	IMod : IModule;
END_VAR
// set up station
ModuleNb := 1;
Module := E_Module.eModule_M001;
Name := stTextListGlobal.stText_M001_Name;

IMod := SUPER^.M_Init()
			  .M_InitEvents(TC_Events.ModuleM010EventClass.InfoEvent,
	  				  		TC_Events.ModuleM010EventClass.WarningEvent,
	  				  		TC_Events.ModuleM010EventClass.ErrorEvent);

// set up default IO references
M_SetReferences(IO.stM001_Module_IO);

// init components


P_Plant.M_RegisterModule(IMod);

bInitSettings	:= FALSE;
bInitMonitoring := FALSE;
bInitManual  	:= FALSE;

//aSClearText[EN] := 'Module init done.';
M_Init := IMod;
END_METHOD

METHOD PROTECTED M_Manual
VAR_INST
	iReq : INT;
END_VAR
// manual mode
IF (OpMode <> E_OpMode.eOpMode_manual) THEN
	RETURN;
END_IF
END_METHOD

METHOD PROTECTED M_OpModeChanged : BOOL
VAR_INPUT
END_VAR
(*bBusy := FALSE;

IF eOpMode <> E_OpMode.eOpMode_auto THEN
	sqAuto.Set(0);
END_IF*)
END_METHOD

METHOD INTERNAL M_RegisterStation : E_Module
VAR_INPUT
	Ist : IStation;
END_VAR
aIStaton[ISt.Station] := ISt;
P_Plant.M_RegisterStation(ISt);
M_RegisterStation := eModule;
END_METHOD

METHOD PUBLIC M_Run : BOOL
VAR_INPUT
END_VAR
VAR
	b1stShot				: BOOL := TRUE;
	stModuleStationsInfoRef	: REFERENCE TO ST_MODULE_STATIONS_INFO;
END_VAR
bSafetyOk := P_Safety.SafetyOk;
aIStaton[E_Station.eStation_ST010_OvenA].SafetyOk := P_Safety.SafetyOk;
aIStaton[E_Station.eStation_ST020_OvenB].SafetyOk := P_Safety.SafetyOk;
aIStaton[E_Station.eStation_ST030_Handling].SafetyOk := P_Safety.SafetyOk;
aIStaton[E_Station.eStation_ST040_Storage].SafetyOk := P_Safety.SafetyOk;
aIStaton[E_Station.eStation_ST050_Mould].SafetyOk := P_Safety.SafetyOk;

// call module base (calls station run)
M_Run := SUPER^.M_Run();

M_DynSettings();
M_DynManual();
M_DynMonitoring();

// loop module stations, collect infos
b1stShot := TRUE;
stModuleStationsInfoRef REF= stGlobalModuleInfo.astModuleStationsInfo[eModule];
FOR ii := 0 TO E_Station.eStation_nMaxIdx DO
	IF aIStaton[ii] = 0 THEN
		CONTINUE;
	END_IF
	
	F_AND_REF_EX(stModuleStationsInfoRef.bStation_All_Auto, aIStaton[ii].OpMode = E_OpMode.eOpMode_auto, b1stShot);
	F_OR_REF_EX(stModuleStationsInfoRef.bStation_Any_Step, aIStaton[ii].OpMode = E_OpMode.eOpMode_step, b1stShot);
	F_OR_REF_EX(stModuleStationsInfoRef.bStation_Any_Manual, aIStaton[ii].OpMode = E_OpMode.eOpMode_manual, b1stShot);
	
	F_OR_REF_EX(stModuleStationsInfoRef.bStation_Any_Error, aIStaton[ii].State = E_ComponentState.eComponentState_error, b1stShot);
	F_OR_REF_EX(stModuleStationsInfoRef.bStation_Any_Warning, aIStaton[ii].State = E_ComponentState.eComponentState_warning, b1stShot);
	F_OR_REF_EX(stModuleStationsInfoRef.bStation_Any_Info, aIStaton[ii].State = E_ComponentState.eComponentState_info, b1stShot);
	
	F_AND_REF_EX(stModuleStationsInfoRef.bStation_All_Started, (aIStaton[ii].OpMode = E_OpMode.eOpMode_auto OR aIStaton[ii].OpMode = E_OpMode.eOpMode_step) AND aIStaton[ii].RunCycle, b1stShot);
	F_AND_REF_EX(stModuleStationsInfoRef.bStation_All_Stopped, aIStaton[ii].Stopped, b1stShot);
	F_AND_REF_EX(stModuleStationsInfoRef.bStation_All_InHome, aIStaton[ii].InHome, b1stShot);
	F_OR_REF_EX(stModuleStationsInfoRef.bStation_Any_Homing, aIStaton[ii].Homing, b1stShot);
	
	b1stShot := FALSE;
END_FOR
END_METHOD

METHOD PROTECTED M_Sequence
VAR
END_VAR
// signal mapping (e.g.: enable)
stM001IModule.bRunCycle := RunCycle;

// automatic sequence
CASE sqAuto.Step OF
	
	0:	sqAuto.Info.Set("Warte auf Auto Start");
		IF NOT (RunCycle AND RunStep) THEN RETURN; END_IF
		
		sqAuto.Info.Set("Warte auf GRST");
		//IF sqHome.InHome AND bInHome THEN
			//fbAxisVm.SetPos(0);
			sqHome.InHome := FALSE;
			sqAuto.Step := 10;
		//ELSE
		//	INotiHdl.M_SetNotiDefaultInf(stTextlistGlobal.stText_NG_Stations, Name, stTextlistGlobal.stText_station_not_in_hp, stEmptyText);
		//END_IF
		
	10:	sqAuto.Info.Set("Prüfe Startbedingungen");
		IF NOT RunCycle THEN sqAuto.Step := 900; END_IF				
		CycleStart();		
		sqAuto.Step := 100;
		
	// work
	100: sqAuto.Info.Set("Automatik");
		TransitionLogic();
		IF NOT RunCycle THEN
			sqAuto.Step := 900;
		END_IF
		
	// stop from safety	or error
	800: sqAuto.Info.Set("Fehler/Safety Stop!");
		FOR ii := 0 TO E_Station.eStation_nMaxIdx DO
			IF aIStaton[ii] <> 0 THEN
				aIStaton[ii].RunCycle := FALSE;
			END_IF
		END_FOR
		sqAuto.Step := 900;		
		
	// rdy	
	900: sqAuto.Info.Set("Zyklus beendet");
		CycleEnd();
		sqAuto.Step := 0;

	// error
	1000: sqAuto.Info.Set("Error");
		bStopped := TRUE;
		sqHome.InHome := FALSE;
		bRunHoming := FALSE;

END_CASE
END_METHOD

METHOD INTERNAL M_SetReferences : BOOL
VAR_IN_OUT
	stIoRef : ST_M001_IO;
END_VAR
stIO REF= stIoRef;
M_SetReferences := TRUE;
END_METHOD

METHOD PROTECTED M_Supervision : BOOL
VAR_INPUT
END_VAR
// to be subclassed// chk stopped
IF NOT bRunCycle OR P_Safety.bMachineRequestStop THEN
	IF sqAuto.StepTime > T#20S THEN
		bStopped := TRUE;
	END_IF
END_IF

(*ToDo: // axis
IF fbAxisVm.bError THEN
	SUPER^.M_SetNotification(F_CreateDynTextUn(E_UniqNoti.eUniqNoti_M001_Module_ServoVm),	// id
					Name,																	// group (e.g.: station name)
					fbAxisVm.Name,															// txt1 (e.g.: source)
					fbAxisVmUi.stErrorText,													// txt2 (e.g.: error text)
					fbAxisVmUi.stBmk,														// txt3 (e.g.: BMK)
					E_AlarmPriority.Error,													// prio
					E_NotificationMode.eNotificationMode_Reset,								// notification mode
					E_AlarmStopMode.Stop);													// alarm stop mode
					

					
ELSIF NOT stIO.stIn.bCentrSuctPwrCircBreakerOk THEN
	SUPER^.M_SetNotification(F_CreateDynTextUn(E_UniqNoti.eUniqNoti_M001_CentralSuction),
					Name,
					F_CreateDynTextDefault("Fehler Netz Schutzschalter"),
					fbCentrSuction.Name,
					F_CreateDynTextDefault("BMK=+xyz-"),
					E_AlarmPriority.Error,
					E_NotificationMode.eNotificationMode_Reset,
					E_AlarmStopMode.Stop);
END_IF *)
END_METHOD

/// Reset station logic
{attribute 'object_name' := 'Reset'}
METHOD Reset
VAR
END_VAR
// base logic run
SUPER^.Reset();
END_METHOD

METHOD PRIVATE TransitionLogic : INT
VAR
	hgCmd : ST_St030_Command;
END_VAR
IF NOT Plant.stSt050IMould.bEnableHG THEN
	sqAuto.Info.Set("Wait for HG enable from mould");
	RETURN;
END_IF

// switxh logic by type
CASE Services.stSettings.stProduct_Settings[E_ProductSettings.eProductSettings_ProductType].nValue OF // or use production settings...
	3: hgCmd := GetHgCmd_Type3(); // e.g.: impelemt custom handling command for type 3...
	5: hgCmd := GetHgCmd_Type5(); // e.g.: impelemt custom handling command for type 5...
	6: hgCmd := GetHgCmd_Type6(); // e.g.: impelemt custom handling command for type 6...
ELSE
	
	// default logic
	hgCmd := GetHgCmd_Default();
END_CASE

Plant.stSt030IHandling.CommandRequest := hgCmd;
END_METHOD

END_FUNCTION_BLOCK

// ---- POUs/Plant/_Base/FB_ModuleBase.TcPOU
FUNCTION_BLOCK FB_ModuleBase EXTENDS FB_ComponentBase IMPLEMENTS IModule
VAR_INPUT
	bEmergencyStopOk 	: BOOL;
	bSafetyOk 			: BOOL;
	bEnable 			: BOOL;
	bAutoHome 			: BOOL;		// if its true station will be homed by start button
	iNumberOfStepChains	: INT := 1;	// count of stepchains per station
	iStepChainIndex		: INT; 		// index to link text of choosed stepchain to hmi
END_VAR
VAR_OUTPUT
	nStateColor			: DWORD;	// color for state of module

	bBusy				: BOOL;		// module is busy
	bTransferEnable		: BOOL;		// transfer enable from module
	stTextAuto			: ST_Text;
	stTextHome			: ST_Text;
	
	/// error-stop status
	bAutoStop_Error		: BOOL;
END_VAR
VAR
	stHmiToModule		: REFERENCE TO ST_DefaultHmiToPlc;				// default hmi to module
	stHmiManualIn		: REFERENCE TO ST_HMI_BASE_MODULE_MANUAL_IN;	// hmi manual to module
	stHmiManualOut		: REFERENCE TO ST_HMI_BASE_MODULE_MANUAL_OUT;	// hmi manual from module
	stLocalSettings		: REFERENCE TO ST_ModuleDynSettings;			// dyn. module settings
	stLocalMonitoring	: REFERENCE TO ST_Monitoring_Module;			// dyn. module monitoring
	
	stLocalSettingsBackup	: ST_ModuleDynSettings;	// dyn. module settings
	
	/// - stations of this module -
	aIStaton	: ARRAY[0..E_Station.eStation_nMaxIdx] OF IStation;
	
	nModuleNb	: INT;
	eModule		: E_Module;
	eOpMode		: E_OpMode;
	bStopped	: BOOL := TRUE;
	
	/// enable var's
	bRunCycle, bRunStep, bRunHoming, bInHome : BOOL;

	/// counter
	diCycles				: UDINT; // Zykluszähler
	diLastCycleTime			: UDINT; // letzte Zykluszeit [ms]
	
	tonOpModeOff			: TON;
	fTrigSafetyOk			: F_TRIG;
	rtrigOpModeChanged		: R_TRIG;
	
	rtirgSafetyOpMode_Auto	: R_TRIG;
	rtirgSafetyOpMode_Hand	: R_TRIG;
	rtirgSafetyOpMode_Aus	: R_TRIG;
	
	bInitSettings	: BOOL;
	bInitMonitoring	: BOOL;
	bInitManual		: BOOL;
	
	sb				: FB_StringBuilder;
	sqHome, sqAuto	: FB_SequenceHelperSb;
	localEvents		: ST_DefaultEventClasses;
END_VAR
VAR PERSISTENT
	diTotalCycles	: UDINT; // Zykluszähler
	eOpModeOld		: E_OpMode;
END_VAR

METHOD PROTECTED CycleEnd
VAR_INPUT
END_VAR
diCycles := diCycles + 1;
diTotalCycles := diTotalCycles + 1;
diLastCycleTime := TIME_TO_UDINT(sqAuto.SeqTime);
sqAuto.StopSequence();
bBusy := FALSE;
//bStopped := TRUE;
END_METHOD

METHOD PROTECTED CycleStart
VAR_INPUT
END_VAR
sqAuto.StartSequence();
bBusy := TRUE;
bStopped := FALSE;
END_METHOD

{attribute 'monitoring':='call'}
PROPERTY PUBLIC EmergencyStopOk : BOOL
GET
EmergencyStopOk := bEmergencyStopOk;
END_GET
SET
bEmergencyStopOk := EmergencyStopOk;
END_SET
END_PROPERTY

{attribute 'monitoring':='call'}
PROPERTY PUBLIC Enable : BOOL
GET
Enable := bEnable;
END_GET
SET
bEnable := Enable;
END_SET
END_PROPERTY

{attribute 'monitoring':='call'}
//{attribute 'monitoring' := 'variable'}
PROPERTY PUBLIC EnableManual : BOOL
GET
EnableManual := EnableSummary AND (eOpMode = eOpMode_manual);
END_GET
END_PROPERTY

{attribute 'monitoring':='call'}
//{attribute 'monitoring' := 'variable'}
PROPERTY INTERNAL EnableSummary : BOOL
GET // PUBLIC
EnableSummary := bEnable 
				AND bSafetyOk 
				AND (eOpMode = eOpMode_manual) OR (eOpMode = eOpMode_step) OR (eOpMode = eOpMode_auto);
END_GET
END_PROPERTY

METHOD PUBLIC GetStepChainTest : ST_Text
VAR_INPUT
	Index : INT; // step chain index
END_VAR
// step chain index is ignored in the default implementation -> if multiple step chains are needed, use derived base and override this method. 
GetStepChainTest.nNameId := sqAuto.InfoTextId;
GetStepChainTest.wsName := sqAuto.Info.ToWString();
GetStepChainTest.wsNameId := sqAuto.InfoTextWsId;
END_METHOD

/// Station in Home flag
{attribute 'monitoring':='call'}
PROPERTY InHome : BOOL
GET
InHome := TRUE;
//FOR ii := 0 TO iNumberOfStepChains - 1 DO
	IF NOT sqHome.InHome THEN
		InHome := FALSE;
	END_IF
//END_FOR

bInHome := InHome;
IF InHome THEN
	bRunHoming := FALSE;
END_IF
END_GET
END_PROPERTY

METHOD PROTECTED M_CallObjects : BOOL
VAR_INPUT
END_VAR
// Call objects - to be subclassed
END_METHOD

METHOD PROTECTED M_DynMonitoring : BOOL
VAR_INPUT
END_VAR
// station base signals
stLocalMonitoring.bInHome := bInHome;
stLocalMonitoring.bAuto := bRunStep;
stLocalMonitoring.bBusy := bBusy;
stLocalMonitoring.bError := (eState = E_ComponentState.eComponentState_error);
stLocalMonitoring.bManual := (eOpMode = E_OpMode.eOpMode_manual);
stLocalMonitoring.bTransferEnable := bTransferEnable;
stLocalMonitoring.bWarning := (eState = E_ComponentState.eComponentState_warning);

M_DynMonitoring := TRUE;
END_METHOD

METHOD PROTECTED M_Homing
VAR
END_VAR
// Homing sequence - to be subclassed
END_METHOD

METHOD PUBLIC M_Init : IModule
VAR_INPUT
END_VAR
// set up defaults
Active := TRUE;
Enable := TRUE;
SUPER^.M_InitComponentBase();

// set up station id and name -> to be subclassed... 
//Module := E_Module.eModule_none;
//Name := stTextListGlobal.stText_M000_Name;

sqAuto.SetInfo(Name);
nStateColor := TO_DWORD(STATICS.stColor.White);

stHmiToModule REF= P_HMI_Controller.aStHmiToModule[eModule];
stHmiManualIn REF= HMI.stHmi.stIn.arrStModule[eModule].stManual;
stHmiManualOut REF= HMI.stHmi.stOut.stCommon.arrStModule[eModule].stManual;
stLocalSettings REF= Services.stSettings.stModuleSettings[eModule];
stLocalMonitoring REF= HMI.stHmi.stOut.stCommon.stMonitoring.astMonitoringModule[eModule];

//FOR ii := 0 TO CONST.iMaxIdxLocalStepChain DO
	sqAuto.SetInfo(stTextListGlobal.stText_initialize_station);	// -> to be subclassed, ... 
//END_FOR

M_Init := THIS^;
END_METHOD

METHOD PROTECTED M_InitDynManual : BOOL
VAR_INPUT
	nIndex			: INT;
	stName			: ST_Text;
	stGroup			: ST_Text;
	stType			: ST_Text;
	diObjectIndex	: DINT;
END_VAR
// chk
IF nIndex < 0 OR nIndex > CONST.iMaxIdxObject THEN
	ModuleError.ArgSbAppendRaise('Dyn. manual index out of range.');
	RETURN;
END_IF

stHmiManualOut.stObjects[nIndex].stName := stName;
stHmiManualOut.stObjects[nIndex].stGroup := stGroup;
stHmiManualOut.stObjects[nIndex].stType := stType;
stHmiManualOut.stObjects[nIndex].diObjectIndex := diObjectIndex;

M_InitDynManual := TRUE;
END_METHOD

METHOD PROTECTED M_InitDynManualUi : BOOL
VAR_IN_OUT
	fbManualUi	: FB_ManualUiBase;
END_VAR
VAR
	IManualUi	: I_ManualUi;
	nIx, ix		: INT;
END_VAR
IManualUi := fbManualUi;

// search next free index
nIx := -1;
FOR ix := 0 TO CONST.iMaxIdxObject DO
	IF stHmiManualOut.stObjects[ix].stName.wsName = "" THEN
		nIx := ix;
		EXIT;
	END_IF
END_FOR

IF nIx < 0 THEN
	ModuleError.ArgSbAppendRaise('Next free dyn. manual index not found.');
	RETURN;
END_IF

IManualUi.ObjectIndex := (ModuleNb * 100) + nIx + 1; // create unique object index

M_InitDynManualUi := M_InitDynManual(nIx,			// index 
		IManualUi.Name,								// device name
		Name,										// group -> module name
		stTextListGlobal.stText_ObjectTypeDrive,	// type
		IManualUi.ObjectIndex);						// object index
		
IManualUi.M_SetStateObject(stHmiManualOut.stObjects[nIx]);
END_METHOD

METHOD PROTECTED M_InitDynMonitoringItem : BOOL
VAR_INPUT
	nIndex		: INT;
	wsName		: WSTRING;
	stGroup		: ST_Text;
	eDataType	: E_DataType;
	stUnit		: ST_Text;			
END_VAR
// chk
IF nIndex < 0 OR nIndex > CONST.iMaxIdxMonitoring THEN
	ModuleError.ArgSbAppendRaise('Dyn. monitoring index out of range.');
	RETURN;
END_IF

stLocalMonitoring.astMonitoring[nIndex].stIndex.nNameId := nIndex;
stLocalMonitoring.astMonitoring[nIndex].stIndex.wsNameId := wsName;
stLocalMonitoring.astMonitoring[nIndex].stName := F_CreateDynText(wsName, nIndex);
stLocalMonitoring.astMonitoring[nIndex].eDataType := eDataType;
stLocalMonitoring.astMonitoring[nIndex].stGroup := stGroup;
stLocalMonitoring.astMonitoring[nIndex].stUnit := stUnit;

M_InitDynMonitoringItem := TRUE;
END_METHOD

METHOD PROTECTED M_InitDynSettingsItem : BOOL
VAR_INPUT
	nIndex					: INT;
	wsIndex					: WSTRING;
	stSettGroup				: ST_Text;
	stSettTitle				: ST_Text;
	stSettUnit				: ST_Text;	
	eSettDataType			: E_DataType;	
	fSettValueMin			: REAL;
	fSettValueMax			: REAL;
	// required user level, 0 = none
	nRequiredUserLevel		: INT := 0;	
END_VAR
// chk
IF nIndex < 0 OR nIndex > CONST.iMaxIdxLocalSetting THEN
	ModuleError.ArgSbAppendRaise('Dyn. setting index out of range.');
	RETURN;
END_IF

M_InitDynSettingsItem := F_InitDynDataItem(
							nIndex,
							wsIndex,
							stSettGroup,
							stSettTitle,
							stSettUnit,
							eSettDataType,
							fSettValueMin,
							fSettValueMax,
							// required user level, 0 = none
							nRequiredUserLevel,
							E_RecipeMode.eRecipeMode_ToFrom,
							stLocalSettings.stDynStationSettings);
END_METHOD

METHOD PUBLIC M_InitEvents : IModule
VAR_IN_OUT CONSTANT
	infoEvent,
	warnEvent,
	errorEvent : TcEventEntry;
END_VAR
// create default module alarms
localEvents.Info := infoEvent;
localEvents.Warning := warnEvent;
localEvents.Error := errorEvent;
IEvent.CreateAlarm(infoEvent, FALSE, TcSourceInfo)
	  .CreateAlarm(warnEvent, TRUE, TcSourceInfo)
	  .CreateAlarm(errorEvent, TRUE, TcSourceInfo);

M_InitEvents := THIS^;
END_METHOD

METHOD Public M_InitEx : IModule
VAR_INPUT
	ILogger			: I_Logger;
	IEventHandler	: I_EventHandler;
END_VAR

// set up logger and event handler
SUPER^.M_InitComponentBaseEx(ILogger, IEventHandler);

// set up module name -> to be subclassed... 
stName := stTextListGlobal.stText_M000_Name;

M_InitEx := THIS^;
END_METHOD

METHOD PROTECTED M_Manual
VAR_INPUT
END_VAR
// Manual mode - to be subclassed
END_METHOD

METHOD PROTECTED M_OpModeChanged : BOOL
VAR_INPUT
END_VAR
// to be subclassed
END_METHOD

METHOD PUBLIC M_Run : BOOL
VAR
END_VAR
M_Run := TRUE;

// call component run
SUPER^.Run();

// loop stations of this module
FOR ii := 0 TO E_Station.eStation_nMaxIdx DO
	IF aIStaton[ii] = 0 THEN
		CONTINUE;
	END_IF
	
	aIStaton[ii].EmergencyStopOk := EmergencyStopOk;
	// specific safety area handled in module -> aIStaton[ii].SafetyOk := SafetyOk;
	M_Run := M_Run AND aIStaton[ii].M_Run(); // call station run
END_FOR

// Safety OP-Mode
rtirgSafetyOpMode_Auto(CLK := stHmiToModule.eSafetyOpMode = E_Opmode.eOpMode_auto);
rtirgSafetyOpMode_Hand(CLK := stHmiToModule.eSafetyOpMode = E_Opmode.eOpMode_manual);
rtirgSafetyOpMode_Aus(CLK := stHmiToModule.eSafetyOpMode = E_Opmode.eOpMode_off);

// reset (all or this station)
IF stHmiToModule.bReset THEN
	Reset();
END_IF

// step (all or this station)
// step -> ist bei Auto über die Property immer TRUE
bRunStep := stHmiToModule.bStep;

// start (all or this station)
IF stHmiToModule.bStart OR stHmiToModule.bStep THEN		
	IF NOT bEnable THEN
		ModuleWarning.ArgSbAppendRaise('Kein Enable Signal bei Start');
	ELSIF NOT bSafetyOk THEN
		ModuleWarning.ArgSbAppendRaise('Safety nicht ok bei Start');
		
	// Fehler steht noch an
	ELSIF bAutoStop_Error THEN
		ModuleWarning.ArgSbAppendRaise('Station in Fehlerstatus --> Reset');
		
	// Safety muss in Auto sein
	ELSIF stHmiToModule.eSafetyOpMode <> E_Opmode.eOpMode_auto AND Const.bEnSafetyOpMode THEN
		ModuleWarning.ArgSbAppendRaise('Safety Betriebsart nicht AUTO');
		
	// START
	ELSIF (OpMode = E_Opmode.eOpMode_auto OR OpMode = E_Opmode.eOpMode_step) THEN
		//bRunStep := FALSE;
		bRunCycle := TRUE;
	END_IF
END_IF

// cycle stop (all or this module)
IF stHmiToModule.bStop OR P_Supervision.bCycleStop THEN
	bRunCycle := bRunHoming := FALSE;
END_IF

// fast stop (all or this module)
IF stHmiToModule.bFastStop OR P_Supervision.bFastStop THEN 
	bRunCycle := bRunStep := bRunHoming := FALSE;
END_IF

// set op mode (all or this module)
tonOpModeOff(IN := stHmiToModule.bStop OR stHmiToModule.bFastStop, PT := T#10S);
IF stHmiToModule.bOpModeManual OR stHmiToModule.bOpModeManual OR rtirgSafetyOpMode_Hand.Q THEN
	bRunStep := FALSE;
	bRunCycle := FALSE;
	bRunHoming := FALSE;
	eOpMode := E_OpMode.eOpMode_manual;
ELSIF stHmiToModule.bOpModeAuto OR stHmiToModule.bOpModeAuto OR rtirgSafetyOpMode_Auto.Q THEN
	bRunStep := FALSE;
	bRunCycle := FALSE;
	bRunHoming := FALSE;
	eOpMode := E_OpMode.eOpMode_auto;
ELSIF stHmiToModule.bOpModeStep THEN
	bRunStep := FALSE;
	bRunCycle := FALSE;
	bRunHoming := FALSE;
	eOpMode := E_OpMode.eOpMode_step;
ELSIF tonOpModeOff.Q THEN
	eOpMode := E_OpMode.eOpMode_off;
END_IF
	
IF NOT bEmergencyStopOk THEN
	sqHome.InHome := FALSE;
	sqHome.Step := 0;
	sqAuto.Step := 0;
END_IF

// homing (all or this station)
IF stHmiToModule.bHome OR (stHmiToModule.bStart AND bAutoHome AND NOT sqHome.InHome AND sqHome.Step = 0 AND sqAuto.Step = 0) THEN
	IF NOT bEnable THEN
		ModuleWarning.ArgSbAppendRaise('Kein Enable Signal bei Start Grundstellung');
	ELSIF NOT bSafetyOk THEN
		ModuleWarning.ArgSbAppendRaise('Safety nicht ok bei Start Grundstellung');
		
	// Fehler steht noch an
	ELSIF bAutoStop_Error THEN
		ModuleWarning.ArgSbAppendRaise('Station in Fehlerstatus --> Reset');
	ELSE		
		sqHome.Step := 0;
		sqHome.InHome		:= FALSE;
		bRunCycle			:= FALSE;
		bRunHoming 			:= TRUE;
	END_IF
END_IF

/// Set Module State Color
IF State = eComponentState_error THEN
	nStateColor := STATICS.stColor.Red;
ELSIF bInHome AND (eOpMode = eOpMode_Auto OR eOpMode = eOpMode_Step) THEN	
	nStateColor := STATICS.stColor.LightBlue;
ELSIF bStopped AND (eOpMode = eOpMode_Auto OR eOpMode = eOpMode_Step) THEN
	nStateColor := STATICS.stColor.Blue;									
ELSIF State = eComponentState_running AND (eOpMode = eOpMode_Auto OR eOpMode = eOpMode_Step) THEN
	nStateColor := STATICS.stColor.LimeGreen;					
ELSIF State = eComponentState_running AND eOpMode = eOpMode_manual THEN
	nStateColor := STATICS.stColor.Orange;		
ELSE
	nStateColor := STATICS.stColor.White;
END_IF

//StepChainTextMapping
//stTextAuto := arraSTextAuto[iStepChainIndex];
IF iStepChainIndex >= 0 AND iStepChainIndex <= CONST.iMaxIdxLocalStepChain THEN
	stTextAuto.nNameId := sqAuto.InfoTextId;
	stTextAuto.wsName := WConcat3(TO_WSTRING(sqAuto.Step),": ", sqAuto.Info.ToWString());
	stTextAuto.wsNameId := WConcat3(TO_WSTRING(sqAuto.Step),": ", sqAuto.InfoTextWsId);	
	
	//stTextHome := arraSTextHome[iStepChainIndex];
	stTextHome.nNameId := sqHome.InfoTextId;
	stTextHome.wsName := WConcat3(TO_WSTRING(sqHome.Step), ": ", sqHome.Info.ToWString());
	stTextHome.wsNameId := WConcat3(TO_WSTRING(sqHome.Step),": ", sqHome.InfoTextWsId);	
END_IF

rtrigOpModeChanged(CLK := eOpModeOld <> eOpMode);
IF rtrigOpModeChanged.Q THEN
	eOpModeOld := eOpMode;
	M_OpModeChanged();
END_IF

//call methodes
sqHome.EnableStep := RunStep;
sqHome();
sqAuto.EnableStep := RunStep;
sqAuto();

M_CallObjects();
M_Homing();
M_Sequence();
M_Manual();
M_Supervision();
END_METHOD

METHOD PROTECTED M_Sequence
VAR
END_VAR
// Automatic sequence - to be subclassed
END_METHOD

METHOD PROTECTED M_Supervision : BOOL
VAR_INPUT
END_VAR
// to be subclassed
END_METHOD

PROPERTY Module : E_Module
GET
Module := eModule;
END_GET
SET
eModule := Module;
END_SET
END_PROPERTY

PROPERTY PROTECTED ModuleError : I_EventHandler
GET
// return the event handler
//	prepare string builder w. module info
ModuleError := IEvent.Select(localEvents.Error)
					 .ArgSbInitWs(stName.wsName)
					 .ArgSbAppend(' | ');
END_GET
END_PROPERTY

PROPERTY PROTECTED ModuleInfo : I_EventHandler
GET
// return the event handler
//	prepare string builder w. module info
ModuleInfo := IEvent.Select(localEvents.Info)
					.ArgSbInitWs(stName.wsName)
					.ArgSbAppend(' | ');
END_GET
END_PROPERTY

PROPERTY PUBLIC ModuleNb : INT
GET
ModuleNb := nModuleNb;
END_GET
SET // PUBLIC
nModuleNb := ModuleNb;
END_SET
END_PROPERTY

PROPERTY PROTECTED ModuleWarning : I_EventHandler
GET
// return the event handler
//	prepare string builder w. module info
ModuleWarning := IEvent.Select(localEvents.Warning)
					   .ArgSbInitWs(stName.wsName)
					   .ArgSbAppend(' | ');
END_GET
END_PROPERTY

/// Station OP Mode
{attribute 'monitoring':='call'}
PROPERTY OpMode : E_OpMode
GET
OpMode := eOpMode;
END_GET
END_PROPERTY

{attribute 'monitoring':='call'}
PROPERTY PUBLIC RunCycle : BOOL
GET // PUBLIC
RunCycle := bRunCycle;
END_GET
SET // PUBLIC
bRunCycle := RunCycle;
END_SET
END_PROPERTY

{attribute 'monitoring':='variable'}
PROPERTY PUBLIC RunStep : BOOL
GET
VAR
	sMsg : WSTRING(255);
END_VAR
// Rückgabe
RunStep := EnableSummary AND
			NOT bAutoStop_Error AND
			((bRunStep AND eOpMode = eOpMode_step) OR
			(eOpMode = eOpMode_auto));
END_GET
END_PROPERTY

{attribute 'monitoring':='call'}
PROPERTY PUBLIC SafetyOk : BOOL
GET
SafetyOk := bSafetyOk;
END_GET
SET
bSafetyOk := SafetyOk;
END_SET
END_PROPERTY

/// Station stopped
{attribute 'monitoring':='call'}
PROPERTY Stopped : BOOL
GET
Stopped := bStopped;
END_GET
END_PROPERTY

PROPERTY TextAuto : ST_Text
GET
TextAuto := stTextAuto;
END_GET
END_PROPERTY

PROPERTY TextHome : ST_Text
GET
TextHome := stTextHome;
END_GET
END_PROPERTY

END_FUNCTION_BLOCK

// ---- POUs/Plant/ST010_OvenA/FB_St010_OvenA.TcPOU
FUNCTION_BLOCK FB_St010_OvenA EXTENDS FB_StationBase
VAR_INPUT
END_VAR
VAR	
	// IO ref
	stIO			: REFERENCE TO ST_St010_IO;
	
	// station components
	fbAxis 			: FB_AxisDriver;
	fbAxisCh1 		: FB_AxisDriver;
	fbAxisCh2 		: FB_AxisDriver;
	
	// actor UIs, access to: iStatus, fPosition, iVisibleState, ..
	fbAxisUi		: FB_Axis_Ui;
	fbAxisCh1Ui		: FB_Axis_Ui;
	fbAxisCh2Ui		: FB_Axis_Ui;
	
	fbHeatingPlate	: FB_FurnaceDriver;
	
	// instance var's
	bStationDeaktiv	: BOOL;
END_VAR
VAR PERSISTENT
	fPickupPos		: LREAL;
END_VAR

/// 
/// Station 010 function block - Oven A
///

{attribute 'monitoring' := 'call'}
PROPERTY PRIVATE HomeSpeed : LREAL
GET
HomeSpeed := stLocalSettings.stDynStationSettings[E_St010_Settings.eSt010_Settings_HomeSpeed].fValue;
END_GET
END_PROPERTY

{attribute 'monitoring' := 'call'}
PROPERTY PRIVATE JogSpeed : LREAL
GET
JogSpeed := stLocalSettings.stDynStationSettings[E_St010_Settings.eSt010_Settings_JogSpeed].fValue;
END_GET
END_PROPERTY

{attribute 'monitoring' := 'call'}
PROPERTY PRIVATE JogSpeedCh : LREAL
GET
JogSpeedCh := stLocalSettings.stDynStationSettings[E_St010_Settings.eSt010_Settings_JogSpeedCh].fValue;
END_GET
END_PROPERTY

METHOD PROTECTED M_CallObjects : BOOL
VAR
END_VAR
//Heating Plate
fbHeatingPlate.Run();

// axis + UI
fbAxis.TorqueLimit := 1000;
fbAxis(
	bEnable := SafetyOk AND NOT fbAxisUi.stAxisManager.bDisable,
	bEnablePos := stSt030IHandling.bEnableOvenAxis OR fbAxisUi.stAxisManager.bDisableSoftLimits,
	bEnableNeg := stSt030IHandling.bEnableOvenAxis OR fbAxisUi.stAxisManager.bDisableSoftLimits
);
fbAxisUi(
	bInHome := bInHome,
	fbAxis := fbAxis,
	fVelocity := JogSpeed,
	diSelectedObjectIndex := stHmiManualIn.diSelectedObjectIndex,
	stHMIControlIn := stHmiManualIn.stManualAxis,
	stHMIControlOut := stHmiManualOut.stManualAxis,
	bJogP := stHmi.stIn.stSt010.bJogUp,
	bJogN := stHmi.stIn.stSt010.bJogDown,
	bEnableManual := EnableManual);	

// axis CH1 + UI
fbAxisCh1(
	bEnable := SafetyOk AND NOT fbAxisCh1Ui.stAxisManager.bDisable,
	bEnablePos := TRUE,
	bEnableNeg := TRUE,
);
fbAxisCh1Ui(
	bInHome := bInHome,
	fbAxis := fbAxisCh1,
	fVelocity := JogSpeedCh,
	diSelectedObjectIndex := stHmiManualIn.diSelectedObjectIndex,
	stHMIControlIn := stHmiManualIn.stManualAxis,
	stHMIControlOut := stHmiManualOut.stManualAxis,
	bJogP := stHmi.stIn.stSt010.bJogCh1Inside,
	bJogN := stHmi.stIn.stSt010.bJogCh1Ouside,
	bEnableManual := EnableManual);
	
// axis CH2 + UI
fbAxisCh2(
	bEnable := SafetyOk AND NOT fbAxisCh2Ui.stAxisManager.bDisable,
	bEnablePos := TRUE,
	bEnableNeg := TRUE,
);
fbAxisCh2Ui(
	bInHome := bInHome,
	fbAxis := fbAxisCh2,
	fVelocity := JogSpeedCh,
	diSelectedObjectIndex := stHmiManualIn.diSelectedObjectIndex,
	stHMIControlIn := stHmiManualIn.stManualAxis,
	stHMIControlOut := stHmiManualOut.stManualAxis,
	bJogP := stHmi.stIn.stSt010.bJogCh2Inside,
	bJogN := stHmi.stIn.stSt010.bJogCh2Ouside,
	bEnableManual := EnableManual);

// HMI : switch between jo modes
//(IF stHmi.stIn.stSt010.bJog THEN
//(	fbAxisUi.ManualMode :=  SEL(stHmi.stIn.stSt010.bSpeed, E_ManualMode.eManualMode_Jog01, E_ManualMode.eManualMode_Jog1);
//(	fbAxisCh1Ui.ManualMode :=  SEL(stHmi.stIn.stSt010.bSpeed, E_ManualMode.eManualMode_Jog01, E_ManualMode.eManualMode_Jog1);
//(	fbAxisCh2Ui.ManualMode :=  SEL(stHmi.stIn.stSt010.bSpeed, E_ManualMode.eManualMode_Jog01, E_ManualMode.eManualMode_Jog1);
//(ELSE
//(	fbAxisUi.ManualMode :=    eManualMode_Tippen ;// SEL(stHmi.stIn.stSt010.bSpeed, E_ManualMode.eManualMode_Tippen, E_ManualMode.eManualMode_TippFast);
//(	fbAxisCh1Ui.ManualMode := eManualMode_Tippen;//	SEL(stHmi.stIn.stSt010.bSpeed, E_ManualMode.eManualMode_TippSlow, E_ManualMode.eManualMode_TippFast);
//(	fbAxisCh2Ui.ManualMode := eManualMode_Tippen;//	SEL(stHmi.stIn.stSt010.bSpeed, E_ManualMode.eManualMode_TippSlow, E_ManualMode.eManualMode_TippFast);
//(END_IF	
	
	
// run trolley logic
//Plant.stSt010IOvenA.Trolley.Update();
END_METHOD

METHOD INTERNAL M_DynManual : BOOL
VAR_INPUT
END_VAR
IF NOT bInitManual THEN
	bInitManual := TRUE;
	MEMSET(ADR(stHmiManualOut.stObjects), 0, SIZEOF(stHmiManualOut.stObjects)); // reset
	
	M_InitDynManualUi(fbAxisUi);
	M_InitDynManualUi(fbAxisCh1Ui);
	M_InitDynManualUi(fbAxisCh2Ui);
	
	fbAxisUi.M_TargetListClear();
	fbAxisUi.M_TargetListAddItem(F_CreateDynText("Home pos", 0), 15);
END_IF
END_METHOD

METHOD PROTECTED M_DynMonitoring : BOOL
VAR_INPUT
END_VAR
M_DynMonitoring := SUPER^.M_DynMonitoring();

// init
IF NOT bInitMonitoring THEN
	bInitMonitoring := TRUE;
	MEMSET(ADR(stLocalMonitoring), 0, SIZEOF(stLocalMonitoring)); // reset
	
	M_InitDynMonitoringItem(0, 								// monitoring index 
							"Achse Position", 				// name
							Name, 							// group (station name)
							E_DataType.eDataType_lreal, 	// data type							
							stTextListGlobal.stText_mm);	// unit	

	M_InitDynMonitoringItem(1, "Achse Geschwindigkeit", Name, E_DataType.eDataType_lreal, stTextListGlobal.stText_mms);
	M_InitDynMonitoringItem(2, "Achse Drehmoment", Name, E_DataType.eDataType_lreal, stTextListGlobal.stText_percent);
	
	M_InitDynMonitoringItem(4, "Achse CH1 Position", Name, E_DataType.eDataType_lreal, stTextListGlobal.stText_mm);
	M_InitDynMonitoringItem(5, "Achse CH1 Geschwindigkeit", Name, E_DataType.eDataType_lreal, stTextListGlobal.stText_mms);
	M_InitDynMonitoringItem(6, "Achse CH1 Drehmoment", Name, E_DataType.eDataType_lreal, stTextListGlobal.stText_percent);
	
	M_InitDynMonitoringItem(8, "Achse CH2 Position", Name, E_DataType.eDataType_lreal, stTextListGlobal.stText_mm);
	M_InitDynMonitoringItem(9, "Achse CH2 Geschwindigkeit", Name, E_DataType.eDataType_lreal, stTextListGlobal.stText_mms);
	M_InitDynMonitoringItem(10, "Achse CH2 Drehmoment", Name, E_DataType.eDataType_lreal, stTextListGlobal.stText_percent);
END_IF

// live value mapping 

// axis
stLocalMonitoring.astMonitoring[0].fValue := fbAxis.Position;
stLocalMonitoring.astMonitoring[1].fValue := fbAxis.Velocity;
stLocalMonitoring.astMonitoring[2].fValue := fbAxis.Torque;

// axis ch1
stLocalMonitoring.astMonitoring[4].fValue := fbAxisCh1.Position;
stLocalMonitoring.astMonitoring[5].fValue := fbAxisCh1.Velocity;
stLocalMonitoring.astMonitoring[6].fValue := fbAxisCh1.Torque;

// axis ch2
stLocalMonitoring.astMonitoring[8].fValue := fbAxisCh2.Position;
stLocalMonitoring.astMonitoring[9].fValue := fbAxisCh2.Velocity;
stLocalMonitoring.astMonitoring[10].fValue := fbAxisCh2.Torque;

// hmi value mapping
//HMI.stHmi.stOut.stSt010.Trolley := stSt010IOvenA.Trolley.stTrolley;
END_METHOD

METHOD INTERNAL M_DynSettings : BOOL
VAR_INPUT
END_VAR
// init station settings
IF NOT bInitSettings THEN
	bInitSettings := TRUE;
	stLocalSettingsBackup := stLocalSettings; // backup
	MEMSET(ADR(stLocalSettings), 0, SIZEOF(stLocalSettings)); // reset
	
	Services.stSettings.stTrolley.CarrierConfig := Services.stSettings.stCarrier;
	stSt010IOvenA.Trolley.Config := Services.stSettings.stTrolley;
	stSt010IOvenA.Trolley.InitialStatus := eTcaWorkpieceStatus.laserProcessDone;
	stSt010IOvenA.Trolley.RequestStatus := eTcaWorkpieceStatus.castingProcessDone;
	stSt010IOvenA.Trolley.ApplyConfig();
	stSt010IOvenA.Trolley.FillWithInitialCarriers();
			
	M_InitDynSettingsItem(E_St010_Settings.eSt010_Settings_Station_Deaktiv,	// settings index
		TO_WSTRING(E_St010_Settings.eSt010_Settings_Station_Deaktiv),		// settings wsIndex
		Name,																// group
		stTextListGlobal.stText_DeactivateStation,							// name
		stTextListGlobal.stText_bool, E_DataType.eDataType_bool,			// unit & data type
		0, 1, 6);															// min, max & user level

	M_InitDynSettingsItem(E_St010_Settings.eSt010_Settings_Autohome,
		TO_WSTRING(E_St010_Settings.eSt010_Settings_Autohome),
		Name,
		stTextListGlobal.stText_AutoHome,
		stTextListGlobal.stText_bool, E_DataType.eDataType_bool,
		0, 1, 3);
		
	M_InitDynSettingsItem(E_St010_Settings.eSt010_Settings_HomeSpeed,
		TO_WSTRING(E_St010_Settings.eSt010_Settings_HomeSpeed),
		Name,
		F_CreateDynTextDefault("Homegeschwindigkeit Servoachse"),
		stTextListGlobal.stText_mms, E_DataType.eDataType_lreal,
		0, 50, 3);
		
	M_InitDynSettingsItem(E_St010_Settings.eSt010_Settings_JogSpeed,
		TO_WSTRING(E_St010_Settings.eSt010_Settings_JogSpeed),
		Name,
		F_CreateDynTextDefault("Tippgeschwindigkeit Servoachse"),
		stTextListGlobal.stText_mms, E_DataType.eDataType_lreal,
		0, 50, 3);
		
	M_InitDynSettingsItem(E_St010_Settings.eSt010_Settings_WorkSpeed,
		TO_WSTRING(E_St010_Settings.eSt010_Settings_WorkSpeed),
		Name,
		F_CreateDynTextDefault("Automatik-Geschwindigkeit Servoachse"),
		stTextListGlobal.stText_mms, E_DataType.eDataType_lreal,
		0, 500, 3);
		
	M_InitDynSettingsItem(E_St010_Settings.eSt010_Settings_JogSpeedCh,
		TO_WSTRING(E_St010_Settings.eSt010_Settings_JogSpeedCh),
		Name,
		F_CreateDynTextDefault("Tippgeschwindigkeit Servoachse CH"),
		stTextListGlobal.stText_mms, E_DataType.eDataType_lreal,
		0, 50, 3);
		
	M_InitDynSettingsItem(E_St010_Settings.eSt010_Settings_WorkSpeedCh,
		TO_WSTRING(E_St010_Settings.eSt010_Settings_WorkSpeedCh),
		Name,
		F_CreateDynTextDefault("Automatik-Geschwindigkeit Servoachse CH"),
		stTextListGlobal.stText_mms, E_DataType.eDataType_lreal,
		0, 500, 3);

	M_InitDynSettingsItem(E_St010_Settings.eSt010_Settings_AxisRefPos,
		TO_WSTRING(E_St010_Settings.eSt010_Settings_AxisRefPos),
		Name,
		F_CreateDynTextDefault("Referenzposition Achse Ofen"),
		stTextListGlobal.stText_m, E_DataType.eDataType_lreal,
		0, 3000, 6);
		
	M_InitDynSettingsItem(E_St010_Settings.eSt010_Settings_PosHome,
		TO_WSTRING(E_St010_Settings.eSt010_Settings_PosHome),
		Name,
		F_CreateDynTextDefault("Homeposition Servoachse"),
		stTextListGlobal.stText_mm, E_DataType.eDataType_lreal,
		0, 5000, 3);
		
	M_InitDynSettingsItem(E_St010_Settings.eSt010_Settings_PosWork,
		TO_WSTRING(E_St010_Settings.eSt010_Settings_PosWork),
		Name,
		F_CreateDynTextDefault("Mitnehmerposition unteres Segment"),
		stTextListGlobal.stText_mm, E_DataType.eDataType_lreal,
		0, 5000, 3);
		
	M_InitDynSettingsItem(E_St010_Settings.eSt010_Settings_PosHomeCh,
		TO_WSTRING(E_St010_Settings.eSt010_Settings_PosHomeCh),
		Name,
		F_CreateDynTextDefault("Homeposition Servoachse CH"),
		stTextListGlobal.stText_mm, E_DataType.eDataType_lreal,
		0, 500, 3);
		
	M_InitDynSettingsItem(E_St010_Settings.eSt010_Settings_PosWorkCh,
		TO_WSTRING(E_St010_Settings.eSt010_Settings_PosWorkCh),
		Name,
		F_CreateDynTextDefault("Arbeitsposition Servoachse CH"),
		stTextListGlobal.stText_mm, E_DataType.eDataType_lreal,
		0, 500, 3);
		
	M_InitDynSettingsItem(E_St010_Settings.eSt010_Settings_OvenFixPartHeight,
		TO_WSTRING(E_St010_Settings.eSt010_Settings_OvenFixPartHeight),
		Name,
		F_CreateDynTextDefault("Festteilhöhe"),
		stTextListGlobal.stText_mm, E_DataType.eDataType_lreal,
		0, 500, 3);
		
	M_InitDynSettingsItem(E_St010_Settings.eSt010_Settings_OvenSegmentHeight,
		TO_WSTRING(E_St010_Settings.eSt010_Settings_OvenSegmentHeight),
		Name,
		F_CreateDynTextDefault("Segmenthöhe"),
		stTextListGlobal.stText_mm, E_DataType.eDataType_lreal,
		0, 500, 3);		
		
	M_InitDynSettingsItem(E_St010_Settings.eSt010_Settings_OvenMiddlePointX,
		TO_WSTRING(E_St010_Settings.eSt010_Settings_OvenMiddlePointX),
		Name,
		F_CreateDynTextDefault("Mittelpunnkt in X-Richtung"),
		stTextListGlobal.stText_mm, E_DataType.eDataType_lreal,
		0, 500, 3);
		
	M_InitDynSettingsItem(E_St010_Settings.eSt010_Settings_OvenOffsetY,
		TO_WSTRING(E_St010_Settings.eSt010_Settings_OvenOffsetY),
		Name,
		F_CreateDynTextDefault("Y-Offset Ofen"),
		stTextListGlobal.stText_mm, E_DataType.eDataType_lreal,
		0, 500, 3);

	M_InitDynSettingsItem(E_St010_Settings.eSt010_Settings_OvenPickUpDepthZ,
		TO_WSTRING(E_St010_Settings.eSt010_Settings_OvenPickUpDepthZ),
		Name,
		F_CreateDynTextDefault("Oven Pick up Depth Z"),
		stTextListGlobal.stText_mm, E_DataType.eDataType_lreal,
		0, 5000, 3);
		
		
	M_InitDynSettingsItem(E_St010_Settings.eSt010_Settings_XPosRp1,	// Teach-Position, Ofen 2, RP 1
		TO_WSTRING(E_St010_Settings.eSt010_Settings_XPosRp1),
		Name,
		F_CreateDynTextDefault("Teach-Position, Ofen 2, RP 1 X"),
		stTextListGlobal.stText_mm, E_DataType.eDataType_lreal,
		0, 5000, 3);
	M_InitDynSettingsItem(E_St010_Settings.eSt010_Settings_YPosRp1,
		TO_WSTRING(E_St010_Settings.eSt010_Settings_YPosRp1),
		Name,
		F_CreateDynTextDefault("Teach-Position, Ofen 2, RP 1 Y"),
		stTextListGlobal.stText_mm, E_DataType.eDataType_lreal,
		0, 3000, 3);
	M_InitDynSettingsItem(E_St010_Settings.eSt010_Settings_ZPosRp1,
		TO_WSTRING(E_St010_Settings.eSt010_Settings_ZPosRp1),
		Name,
		F_CreateDynTextDefault("Teach-Position, Ofen 2, RP 1 Z"),
		stTextListGlobal.stText_mm, E_DataType.eDataType_lreal,
		0, 1000, 3);
		
	M_InitDynSettingsItem(E_St010_Settings.eSt010_Settings_XPosRp2,	// Teach-Position, Ofen 2, RP 2
		TO_WSTRING(E_St010_Settings.eSt010_Settings_XPosRp2),
		Name,
		F_CreateDynTextDefault("Teach-Position, Ofen 2, RP 2 X"),
		stTextListGlobal.stText_mm, E_DataType.eDataType_lreal,
		0, 5000, 3);
	M_InitDynSettingsItem(E_St010_Settings.eSt010_Settings_YPosRp2,
		TO_WSTRING(E_St010_Settings.eSt010_Settings_YPosRp2),
		Name,
		F_CreateDynTextDefault("Teach-Position, Ofen 2, RP 2 Y"),
		stTextListGlobal.stText_mm, E_DataType.eDataType_lreal,
		0, 3000, 3);
	M_InitDynSettingsItem(E_St010_Settings.eSt010_Settings_ZPosRp2,
		TO_WSTRING(E_St010_Settings.eSt010_Settings_ZPosRp2),
		Name,
		F_CreateDynTextDefault("Teach-Position, Ofen 2, RP 2 Z"),
		stTextListGlobal.stText_mm, E_DataType.eDataType_lreal,
		0, 1000, 3);
		
	// restore values
	F_RestoreSettingValues(stLocalSettings.stDynStationSettings, stLocalSettingsBackup.stDynStationSettings);
END_IF

// map current settings values
bStationDeaktiv := stLocalSettings.stDynStationSettings[E_St010_Settings.eSt010_Settings_Station_Deaktiv].bValue;
bAutoHome := stLocalSettings.stDynStationSettings[E_St010_Settings.eSt010_Settings_Autohome].bValue;
END_METHOD

METHOD PROTECTED M_Homing
VAR
	stHomPrm : ST_AxisHomingParameter;
END_VAR
// Homing sequence
CASE sqHome.Step OF
	
	0:	
		sqHome.Info.Set("Warte auf GRST Start");
			
		IF RunStep AND NOT sqHome.InHome AND bRunHoming THEN
			stSt010IOvenA.bResponseOpn := FALSE;
			bBusy := TRUE;
			sqAuto.Step := 0;
			sqHome.StartSequence()
				  .Step := 10;
		END_IF

	10:
		sqHome.Info.Set("Grundstellungsfahrt aktiv");
		IF P_Safety.bMachineRequestStop THEN
			sqHome.Info.Set("Anforderung Stop aktiv");
		ELSIF NOT SafetyOk THEN
			sqHome.Info.Set("Sicherheit nicht ok");
			
		ELSIF NOT fbAxis.Operational THEN
			sqHome.Info.Set("Antrieb Ofen nicht bereit");			
		ELSIF fbAxis.Moving THEN
			fbAxis.Halt();
			sqHome.Info.Set("Antrieb Ofen nicht gestoppt");
		ELSIF NOT stSt030IHandling.bEnableOvenAxis THEN
			sqHome.Info.Set("Warte auf Fahrfreigabe vom HG");
			
		ELSIF NOT fbAxisCh1.Operational THEN
			sqHome.Info.Set("Antrieb Ofen CH1 nicht bereit");
		ELSIF fbAxisCh1.Moving THEN
			fbAxisCh1.Halt();
			sqHome.Info.Set("Antrieb Ofen CH1 nicht gestoppt");
			
		ELSIF NOT fbAxisCh2.Operational THEN
			sqHome.Info.Set("Antrieb Ofen CH2 nicht bereit");
		ELSIF fbAxisCh2.Moving THEN
			fbAxisCh2.Halt();
			sqHome.Info.Set("Antrieb Ofen CH2 nicht gestoppt");

		ELSIF bRunHoming THEN
			sqHome.Step := 15;
		END_IF
		
	15:	sqHome.Info.Set("Prüfe Status");
		IF F_TargetWindowReached(fbAxisCh1.Position, PosHomeCh, chAxisPosTol) AND 
		   F_TargetWindowReached(fbAxisCh2.Position, PosHomeCh, chAxisPosTol) THEN
			sqHome.SetStep(20);
		ELSIF fbAxis.Homed THEN
			sqHome.SetStep(16); // close segment
		ELSE
			StationError.ArgSbAppendRaise('Segmenttor manuell schließen!');
		END_IF
		
	16: sqHome.Info.Set("Start Achse zu Arbeitspos.");
		fbAxis.MoveAbsExVel(fPickupPos, WorkSpeed);
		sqHome.Step := 17;
		
	17: sqHome.Info.Set("Warte auf Achse in Arbeitspos");
		IF fbAxis.TargetReached() THEN
			sqHome.SetStep(20); // ch axis back
		END_IF
		
	20:
		sqHome.Info.Set("Grundstellungsfahrt aktiv Achse CH1 auf Homepos.");
		fbAxisCh1.MoveAbsExVel(PosHomeCh, WorkSpeedCh);
		sqHome.Step := 25;
		
	25:
		sqHome.Info.Set("Warte auf Achse CH1 in Homeposition");
		IF fbAxisCh1.TargetWindowReached(chAxisPosTol) THEN
			sqHome.Step := 30;
		END_IF
		
	30:
		sqHome.Info.Set("Grundstellungsfahrt aktiv Achse CH2 auf Homepos.");
		fbAxisCh2.MoveAbsExVel(PosHomeCh, WorkSpeedCh);
		sqHome.Step := 35;
		
	35:
		sqHome.Info.Set("Warte auf Achse CH2 in Homeposition");
		IF fbAxisCh2.TargetWindowReached(chAxisPosTol) THEN
			sqHome.Step := 40;
		END_IF
	
	40:
		sqHome.Info.Set("Prüfe Achskalibrierung");
		IF fbAxis.Homed THEN
			sqHome.Step := 50;
		ELSE
			sqHome.Step := 42;
		END_IF
		
	42:
		sqHome.Info.Set("Starte Achskalibrierung");
		IF RunStep THEN
			stHomPrm.fPosition := OvenRefPos;
			stHomPrm.stOptions.SearchDirection := MC_Direction.MC_Negative_Direction;
			stHomPrm.stOptions.SyncDirection := MC_Direction.MC_Positive_Direction;
			stHomPrm.stOptions.SearchVelocity := 8;
			stHomPrm.stOptions.SyncVelocity := 4;
			fbAxis.HomeEx(stHomPrm);
			sqHome.Step := 44;
		END_IF
		
	44:
		sqHome.Info.Set("Warte auf Achskalibrierung fertig");
		fbAxis.bCalibrationCam := stIO.stIn.bRefpos;
		IF fbAxis.Homed THEN
			sqHome.Step := 50;
		END_IF
		
	50:
		sqHome.Info.Set("Grundstellungsfahrt aktiv Achse auf Homepos.");
		fbAxis.MoveAbsExVel(PosHome, HomeSpeed);
		sqHome.Step := 60;
		
	60:
		sqHome.Info.Set("Warte auf Achse in Homeposition");
		IF fbAxis.TargetReached() THEN
			sqHome.Step := 100;
		END_IF
		
	100:
		sqHome.Info.Set("Grundstellungsfahrt aktiv");
		sqHome.Step := 1000;

	//	homing done			
	1000:
		sqHome.Info.Set("Grundstellung erreicht");
		IF sqHome.StepTime > T#1S THEN
			bBusy:=FALSE;
			sqHome.InHome := TRUE;
			bStopped := TRUE;
			bRunHoming := FALSE;
			sqAuto.Step := 0;
			sqHome.StopSequence()
				  .Step := 0;
		END_IF
END_CASE
END_METHOD

METHOD PUBLIC M_Init : IStation
VAR_INPUT
END_VAR
VAR
	Ist : IStation;
END_VAR
// set up station
StationNb := 10;
Station := E_Station.eStation_ST010_OvenA; // ID & name 1st!
Name := F_CreateDynTextEx(1, "ST010_OvenA", "ST010 Ofen A");

Ist := SUPER^.M_Init()
			 .InitEvents(TC_Events.ST010EventClass.InfoEvent,
	  		       		 TC_Events.ST010EventClass.WarningEvent,
	  				  	 TC_Events.ST010EventClass.ErrorEvent);

// set up default IO references
M_SetReferences(IO.st010_OvenA_IO);

// init components

// Axis
fbAxisUi.stBmk := F_CreateDynTextDefault("BMK=A03.ST10.M01-");
fbAxisUi.stUnit := F_CreateDynTextDefault("mm");
fbAxisUi.stAxisManager.bEnablePosSet := TRUE;
fbAxisUi.stAxisManager.bSetCalibrationVisible := TRUE;
fbAxisUi.stAxisManager.bResetCalibrationVisible := TRUE;
fbAxis.AxisId := TO_INT(E_Axis.eAxis_OvenA);
fbAxis.Active := TRUE;
fbAxis.Name := F_CreateDynTextEx(1, "ServoOvenA", "Servoachse Ofen A");
fbAxis.AxisType := E_AxisType.AX5xxx;
//fbAxis.DefaultParameter := F_GetDefaultMotionParameter(eMainState_setup);
fbAxis.SetAxisReference(NcIO.stAxis_ST010_OvenA, NcIO.stAxis_ST010_OvenA_IO.stIn, NCIO.stAxis_ST010_OvenA_IO.stOut);

// Axis CH1
fbAxisCh1Ui.stBmk := F_CreateDynTextDefault("BMK=A03.ST10.M02-");
fbAxisCh1Ui.stUnit := F_CreateDynTextDefault("mm");
fbAxisCh1Ui.stAxisManager.bEnablePosSet := TRUE;
fbAxisCh1.AxisId := TO_INT(E_Axis.eAxis_OvenA_CH1);
fbAxisCh1.Active := TRUE;
fbAxisCh1.Name := F_CreateDynTextEx(1, "ServoOvenACh1", "Servoachse Ofen A CH1");
fbAxisCh1.AxisType := E_AxisType.AX5xxx;
//fbAxisCh1.DefaultParameter := F_GetDefaultMotionParameter(eMainState_setup);
fbAxisCh1.SetAxisReference(NcIO.stAxis_ST010_OvenACh1, NcIO.stAxis_ST010_OvenACh1_IO.stIn, NCIO.stAxis_ST010_OvenACh1_IO.stOut);

// Axis CH2
fbAxisCh2Ui.stBmk := F_CreateDynTextDefault("BMK=A03.ST10.M03-");
fbAxisCh2Ui.stUnit := F_CreateDynTextDefault("mm");
fbAxisCh2Ui.stAxisManager.bEnablePosSet := TRUE;
fbAxisCh2.AxisId := TO_INT(E_Axis.eAxis_OvenA_CH2);
fbAxisCh2.Active := TRUE;
fbAxisCh2.Name := F_CreateDynTextEx(1, "ServoOvenACh2", "Servoachse Ofen A CH2");
fbAxisCh2.AxisType := E_AxisType.AX5xxx;
//fbAxisCh2.DefaultParameter := F_GetDefaultMotionParameter(eMainState_setup);
fbAxisCh2.SetAxisReference(NcIO.stAxis_ST010_OvenACh2, NcIO.stAxis_ST010_OvenACh2_IO.stIn, NCIO.stAxis_ST010_OvenACh2_IO.stOut);

// register station in it's module
eParent := fbModul001.M_RegisterStation(Ist);

bInitSettings	:= FALSE;
bInitMonitoring := FALSE;
bInitManual  	:= FALSE;

//aSClearText[EN] := 'Station init done.';
M_Init := Ist;

//IF Firstrun THEN
//	Firstrun := FALSE;
//	
//	// init Settings
//	GlobalSetting.Carrier.CoordinateFirstWorkpiece.fX := 32;
//	GlobalSetting.Carrier.CoordinateFirstWorkpiece.fY := 60;
//	GlobalSetting.Carrier.Dimension.fX := 400;
//	GlobalSetting.Carrier.Dimension.fY := 600;
//	GlobalSetting.Carrier.Layout := eTcaCarrierLayout.Layout1;
//	GlobalSetting.Carrier.PositionsInColumn := 9;
//	GlobalSetting.Carrier.PositionsInRow := 7;
//	GlobalSetting.Carrier.ColumnDistance := 56;		// X Direction
//	GlobalSetting.Carrier.RowDistance := 60;		// Y Direction
//	
//	GlobalSetting.Trolley.CarrierDistance := 80;
//	GlobalSetting.Trolley.NumberOfCarriers := 40;
//	GlobalSetting.Trolley.RackOrigin.fX := 0;
//	GlobalSetting.Trolley.RackOrigin.fY := 278;
//	GlobalSetting.Trolley.RackDivision := 443;
//
//END_IF
//
//IF apply THEN
//	apply := FALSE;
//	
//	GlobalSetting.Trolley.CarrierConfig := GlobalSetting.Carrier;
//	// Init Items
//	_Trolley.Config := GlobalSetting.Trolley;
//	//_Trolley.Config.CarrierConfig := GlobalSetting.Carrier;
//	_Trolley.InitialStatus := eTcaWorkpieceStatus.laserProcessDone;
//	_Trolley.RequestStatus := eTcaWorkpieceStatus.castingProcessDone;
//	_Trolley.ApplyConfig();
//	_Trolley.FillWithInitialCarriers();
//	
//	_Trolley2.Config := GlobalSetting.Trolley;
//	//_Trolley2.Config.CarrierConfig := GlobalSetting.Carrier;	
//	_Trolley2.InitialStatus := eTcaWorkpieceStatus.laserProcessDone;
//	_Trolley2.RequestStatus := eTcaWorkpieceStatus.castingProcessDone;
//	_Trolley2.ApplyConfig();
//	_Trolley2.FillWithEmptyCarriers();
//	
//	
//	_Carrier.Config := GlobalSetting.Carrier;
//	_Carrier.ApplyConfig();
//	        
//	_Carrier2.Config := GlobalSetting.Carrier;
//	_Carrier2.ApplyConfig();
//	
//END_IF
END_METHOD

METHOD PROTECTED M_Manual
VAR
END_VAR

// station must be stopped!			manual mode
IF RunCycle OR NOT bStopped THEN //(OpMode <> E_OpMode.eOpMode_manual) THEN
	RETURN;
END_IF

stSt010IOvenA.Trolley.ServiceMode();



//IF stHmiInOut.stSt010.Command = E_HMI_TR_CMD.eHmiTrCmd_none AND_THEN 
//   stHmiInOut.stSt010.PlCmd.Command <> E_HMI_PL_CMD.eHmiPlCmd_none THEN
//	stHmiInOut.stSt010.Command := E_HMI_TR_CMD.eHmiTrCmd_performPlCmd;
//END_IF
//
//IF stHmiInOut.stSt010.Command = E_HMI_TR_CMD.eHmiTrCmd_performPlCmd THEN
//	RETURN;
//END_IF
//
//stSt010IOvenA.Trolley.PerformHmiCmd(stHmiInOut.stSt010);
END_METHOD

METHOD PROTECTED M_OpModeChanged : BOOL
VAR_INPUT
END_VAR
(*bBusy := FALSE;

IF (eOpMode <> eOpMode_step AND eOpMode <> eOpMode_auto) THEN
	sqAuto.Set(0);
END_IF

fbAxis.Stop();
fbAxisCh1.Stop();
fbAxisCh2.Stop();*)
END_METHOD

METHOD PUBLIC M_Run : BOOL
VAR_INPUT
END_VAR
// check refs valid
IF NOT __ISVALIDREF(stIO) THEN
	RETURN;
END_IF

M_RUN := SUPER^.M_Run();

M_DynSettings();
M_DynManual();
M_DynMonitoring();
END_METHOD

METHOD PROTECTED M_Sequence
VAR
	fTmp : LREAL;
END_VAR
// signal mapping (e.g.: enable)
stSt010IOvenA.bEnableSequence := (sqAuto.Step = 100 AND fbAxis.Operational AND fbAxisCh1.Operational AND fbAxisCh2.Operational) OR
									bStationDeaktiv;

// automatic sequence
CASE sqAuto.Step OF
	
	0:	sqAuto.Info.Set("Warte auf Auto Start");
		IF RunCycle AND RunStep THEN
			//sqAuto.Info.Set("Warte auf GRST");
			//IF sqAuto.InHome AND bInHome THEN
				sqAuto.InHome := FALSE;
				sqAuto.Step := 10;
			//ELSE
			//	StationError.ArgSbAppendWsRaise(stTextlistGlobal.stText_station_not_in_hp);
			//END_IF
		END_IF
		
	10:	sqAuto.Info.Set("Prüfe Startbedingungen");
		IF NOT (fbAxis.Operational AND fbAxis.Homed) THEN
			StationError.ArgSbAppendRaise('Achse nicht bereit');
		ELSIF NOT fbAxisCh1.Operational THEN
			StationError.ArgSbAppendRaise('Achse CH1 nicht bereit');
		ELSIF NOT fbAxisCh2.Operational THEN
			StationError.ArgSbAppendRaise('Achse CH2 nicht bereit');
		ELSE
			CycleStart();
			//stSt010IOvenA.bStorageEnd := FALSE;
			sqAuto.Step := 15;
		END_IF
		
	15:	sqAuto.Info.Set("Prüfe Status");
		IF F_TargetWindowReached(fbAxisCh1.Position, PosHomeCh, chAxisPosTol) AND 
		   F_TargetWindowReached(fbAxisCh2.Position, PosHomeCh, chAxisPosTol) THEN
			sqAuto.SetStep(20);
		ELSE
			sqAuto.SetStep(160); // close segment
		END_IF
		
	20:	sqAuto.Info.Set("Start Achse CH1 auf Homepos.");
		fbAxisCh1.MoveAbsExVel(PosHomeCh, WorkSpeedCh);
		fbAxisCh2.MoveAbsExVel(PosHomeCh, WorkSpeedCh);
		sqAuto.Step := 30;
		
	30:	sqAuto.Info.Set("Warte Achse CH1 in Homeposition");
		IF NOT fbAxisCh1.TargetWindowReached(chAxisPosTol) THEN RETURN; END_IF
		sqAuto.Info.Set("Warte Achse CH2 in Homeposition");
		IF NOT fbAxisCh2.TargetWindowReached(chAxisPosTol) THEN RETURN; END_IF
		sqAuto.SetStep(100);

	// work
	100: sqAuto.Info.Set("Automatik, warte auf Anforderung vom HG");
		IF stSt030IHandling.bReqestOvenA_ChkIndex THEN
			sqAuto.Info.Append(", Index-Check");
			stSt010IOvenA.iConfirmPosition := stSt030IHandling.ActiveCommand.Position;
			stSt010IOvenA.bResponseIsEmptySlot := stSt010IOvenA.Trolley.IsEmptySlotAt(stSt010IOvenA.iConfirmPosition);
			stSt010IOvenA.bResponseChkIndex := TRUE;
			IF stSt030IHandling.bReqestOvenA THEN sqAuto.SetStep(110); END_IF
		END_IF	
		IF RunCycle THEN RETURN; END_IF
		sqAuto.Info.Set("Stop - warte auf Ablauf gestoppt");
		sqAuto.Step := 900;
		
	110: sqAuto.Info.Set("Start Achse zu Arbeitspos.");
		fPickupPos := PosWork;
		fbAxis.MoveAbsExVel(fPickupPos, WorkSpeed);
		sqAuto.Step := 115;
		
	115: sqAuto.Info.Set("Warte auf Achse in Arbeitspos");
		IF fbAxis.TargetReached() THEN
			sqAuto.SetStep(120);
		END_IF
		
	120: sqAuto.Info.Set("Start Achse CH1 zu Arbeitspos.");
		fbAxisCh1.MoveAbsExVel(PosWorkCh, WorkSpeedCh);
		fbAxisCh2.MoveAbsExVel(PosWorkCh, WorkSpeedCh);
		sqAuto.Step := 125;
		
	125: sqAuto.Info.Set("Warte Achse CH1 in Arbeitspos");
		IF fbAxisCh1.TargetWindowReached(chAxisPosTol) THEN
			sqAuto.SetStep(130);
		END_IF
		
	130: sqAuto.Info.Set("Start Achse CH2 zu Arbeitspos.");
		fbAxisCh2.MoveAbsExVel(PosWorkCh, WorkSpeedCh);
		sqAuto.Step := 135;
		
	135: sqAuto.Info.Set("Warte Achse CH2 in Arbeitspos");
		IF fbAxisCh2.TargetWindowReached(chAxisPosTol) THEN
			sqAuto.SetStep(140);
		END_IF
		
	140: sqAuto.Info.Set("Start Achse zu Arbeitspos. offen");
		fTmp := (PosWorkOpn - PosWork);
		IF fTmp > 540 THEN
			sqAuto.Info.Set("Max. Öffnungsweg überschritten: ")
					   .AppendAny(fTmp);
					   
			StationError.ArgSbAppendS(sqAuto.Info.ToString())
						.Raise();
			RETURN;
		END_IF
		fbAxis.MoveAbsExVel(PosWorkOpn, WorkSpeed);
		sqAuto.Step := 145;
		
	145: sqAuto.Info.Set("Warte auf Achse in Arbeitspos. offen");
		IF fbAxis.TargetReached() THEN
			sqAuto.Step := 150;
		END_IF
		
	150: sqAuto.Info.Set("Segment offen, warte auf Anforderung vom HG");
		stSt010IOvenA.bResponseOpn := TRUE;
		IF NOT stSt030IHandling.bReqestOvenA THEN
			stSt010IOvenA.bResponseOpn := FALSE;
			sqAuto.SetStep(160);
		END_IF
		
	160: sqAuto.Info.Set("Start Achse zu Arbeitspos.");
		fbAxis.MoveAbsExVel(fPickupPos, WorkSpeed);
		sqAuto.Step := 165;
		
	165: sqAuto.Info.Set("Warte auf Achse in Arbeitspos");
		IF fbAxis.TargetReached() THEN
			sqAuto.SetStep(170);
		END_IF
		
	170: sqAuto.Info.Set("Start Achse CH1 auf Homepos.");
		fbAxisCh1.MoveAbsExVel(PosHomeCh, WorkSpeedCh);
		fbAxisCh2.MoveAbsExVel(PosHomeCh, WorkSpeedCh);
		sqAuto.Step := 175;
		
	175:	sqAuto.Info.Set("Warte Achse CH1 in Homeposition");
		IF NOT fbAxisCh1.TargetWindowReached(chAxisPosTol) THEN RETURN; END_IF
		sqAuto.Info.Set("Warte Achse CH2 in Homeposition");
		IF NOT fbAxisCh2.TargetWindowReached(chAxisPosTol) THEN RETURN; END_IF
		sqAuto.SetStep(900);
		
	// rdy	
	900: sqAuto.Info.Set("Zyklus beendet");
		CycleEnd();
		sqAuto.Step := 0;	// ch axis back, loop

	// error
	1000: sqAuto.Info.Set("Error");
		bStopped := TRUE;
		sqAuto.InHome := FALSE;
		bRunHoming := FALSE;

END_CASE
END_METHOD

METHOD INTERNAL M_SetReferences : BOOL
VAR_IN_OUT
	stIoRef : ST_St010_IO;
END_VAR
stIO REF= stIoRef;
M_SetReferences := TRUE;

fbHeatingPlate.SetReferences(stIoRef.stHeatingPlateIO);
END_METHOD

METHOD PROTECTED M_Supervision : BOOL
VAR
END_VAR
// chk stopped
IF NOT bRunCycle OR P_Safety.bMachineRequestStop THEN
	IF P_Safety.bMachineRequestStop THEN
		fbAxis.Stop();
	END_IF
	IF sqAuto.StepTime > T#20S THEN
		bStopped := TRUE;
	END_IF
END_IF

// chk requested index
IF stSt030IHandling.bReqestOvenA_ChkIndex THEN
	;// --> confirm chk implemented in M_Sequence, step 100
	//stSt010IOvenA.iConfirmOpnIdxX := stSt030IHandling.ActiveCommand.IndexX;
	//stSt010IOvenA.iConfirmOpnIdxY := stSt030IHandling.ActiveCommand.IndexY;
	//stSt010IOvenA.bResponseEmptyAtIndex := stSt010IOvenA.Trolley.IsEmptySlotAt(stSt010IOvenA.iConfirmOpnIdxX, stSt010IOvenA.iConfirmOpnIdxY);
	//stSt010IOvenA.bResponseChkIndex := TRUE;
ELSE
	stSt010IOvenA.iConfirmPosition := -1;
	stSt010IOvenA.bResponseIsEmptySlot := FALSE;
	stSt010IOvenA.bResponseChkIndex := FALSE;
END_IF

// axis
IF fbAxis.bError THEN
	ReactToComponentError(fbAxisUi, E_EventReaction.Stop);
	
// ch1
ELSIF fbAxisCh1.bError THEN
	ReactToComponentError(fbAxisCh1Ui, E_EventReaction.Stop);
	
// ch2
ELSIF fbAxisCh2.bError THEN
	ReactToComponentError(fbAxisCh2Ui, E_EventReaction.Stop);
	
END_IF
END_METHOD

{attribute 'monitoring' := 'call'}
PROPERTY PRIVATE OvenFixPartHeight : LREAL
GET
OvenFixPartHeight := stLocalSettings.stDynStationSettings[E_St010_Settings.eSt010_Settings_OvenFixPartHeight].fValue;
END_GET
END_PROPERTY

{attribute 'monitoring' := 'call'}
PROPERTY INTERNAL OvenMiddlePointX : LREAL
GET
OvenMiddlePointX := stLocalSettings.stDynStationSettings[E_St010_Settings.eSt010_Settings_OvenMiddlePointX].fValue;
END_GET
END_PROPERTY

{attribute 'monitoring' := 'call'}
PROPERTY INTERNAL OvenOffsetY : LREAL
GET
OvenOffsetY := stLocalSettings.stDynStationSettings[E_St010_Settings.eSt010_Settings_OvenOffsetY].fValue;
END_GET
END_PROPERTY

{attribute 'monitoring' := 'call'}
PROPERTY INTERNAL OvenPickUpDepthZ : LREAL
GET
OvenPickUpDepthZ := stLocalSettings.stDynStationSettings[E_St010_Settings.eSt010_Settings_OvenPickUpDepthZ].fValue;
END_GET
END_PROPERTY

{attribute 'monitoring' := 'call'}
PROPERTY INTERNAL OvenRefPos : LREAL
GET
OvenRefPos := stLocalSettings.stDynStationSettings[E_St010_Settings.eSt010_Settings_AxisRefPos].fValue;
END_GET
END_PROPERTY

{attribute 'monitoring' := 'call'}
PROPERTY PRIVATE OvenSegmentHeight : LREAL
GET
OvenSegmentHeight := stLocalSettings.stDynStationSettings[E_St010_Settings.eSt010_Settings_OvenSegmentHeight].fValue;
END_GET
END_PROPERTY

{attribute 'monitoring' := 'call'}
PROPERTY INTERNAL PosHome : LREAL
GET
PosHome := stLocalSettings.stDynStationSettings[E_St010_Settings.eSt010_Settings_PosHome].fValue;
END_GET
END_PROPERTY

